# B&R Automation Studio project NAELD004C00R10L518F00 (part 12)

#### Act_OptP0930MagConv1FB.st
```iecst
ACTION Act_OptP0930MagConv1FB:

	//Magazine Conveyor
	IF tyP0930MagConv1.tyFB.tyBtnStop.bRtCompl = TRUE THEN
		eMagConv2Clp1Act	:= MagConv2ClpActStop;

		IF p_eMagConv2Clp1Stat = MagConv2ClpActStop AND p_eMagConv2Clp1Status = Done THEN
			eMagConv2Clp1Act	:= MagConv2ClpActIdle;

			tyP0930MagConv1.tyFB.tyBtnEnt.bRtCompl	:= FALSE;
			tyP0930MagConv1.tyFB.tyBtnEnt.bValue	:= FALSE;
			tyP0930MagConv1.tyFB.tyBtnEnt.bRtLk		:= FALSE;

			tyP0930MagConv1.tyFB.tyBtnExit.bRtCompl	:= FALSE;
			tyP0930MagConv1.tyFB.tyBtnExit.bValue	:= FALSE;
			tyP0930MagConv1.tyFB.tyBtnExit.bRtLk	:= FALSE;

			tyP0930MagConv1.tyFB.tyBtnStop.bRtCompl	:= FALSE;
			tyP0930MagConv1.tyFB.tyBtnStop.bValue	:= TRUE;
			tyP0930MagConv1.tyFB.tyBtnStop.bRtLk	:= TRUE;
		END_IF

	ELSIF tyP0930MagConv1.tyFB.tyBtnEnt.bRtCompl = TRUE THEN
		tyP0930MagConv1.tyFB.tyBtnEnt.bValue	:= TRUE;
		tyP0930MagConv1.tyFB.tyBtnEnt.bRtLk		:= TRUE;

		tyP0930MagConv1.tyFB.tyBtnStop.bValue	:= FALSE;
		tyP0930MagConv1.tyFB.tyBtnStop.bRtLk	:= FALSE;

		eMagConv2Clp1Act	:= MagConv2ClpActEnt;

		IF p_eMagConv2Clp1Stat = MagConv2ClpActEnt AND p_eMagConv2Clp1Status = Done THEN
			eMagConv2Clp1Act	:= MagConv2ClpActIdle;

			tyP0930MagConv1.tyFB.tyBtnEnt.bRtCompl	:= FALSE;

			tyP0930MagConv1.tyFB.tyBtnEnt.bValue	:= FALSE;
			tyP0930MagConv1.tyFB.tyBtnEnt.bRtLk		:= FALSE;

			tyP0930MagConv1.tyFB.tyBtnStop.bValue	:= TRUE;
			tyP0930MagConv1.tyFB.tyBtnStop.bRtLk	:= TRUE;
		END_IF

	ELSIF (p_eMagConv2Clp1Stat = MagConv2ClpActPreExit AND p_eMagConv2Clp1Status = Done) THEN
		eMagConv2Clp1Act	:= MagConv2ClpActIdle;

		tyP0930MagConv1.tyFB.tyBtnExit.bRtCompl	:= FALSE;

		tyP0930MagConv1.tyFB.tyBtnExit.bValue	:= FALSE;
		tyP0930MagConv1.tyFB.tyBtnExit.bRtLk	:= FALSE;

		tyP0930MagConv1.tyFB.tyBtnStop.bValue	:= TRUE;
		tyP0930MagConv1.tyFB.tyBtnStop.bRtLk	:= TRUE;

	ELSIF (p_eMagConv2Clp1Stat = MagConv2ClpActExit AND p_eMagConv2Clp1Status = Done) THEN
		eMagConv2Clp1Act	:= MagConv2ClpActIdle;

		tyP0930MagConv1.tyFB.tyBtnExit.bRtCompl	:= FALSE;

		tyP0930MagConv1.tyFB.tyBtnExit.bValue	:= FALSE;
		tyP0930MagConv1.tyFB.tyBtnExit.bRtLk	:= FALSE;

		tyP0930MagConv1.tyFB.tyBtnStop.bValue	:= TRUE;
		tyP0930MagConv1.tyFB.tyBtnStop.bRtLk	:= TRUE;

	ELSIF tyP0930MagConv1.tyFB.tyBtnExit.bRtCompl = TRUE THEN
		tyP0930MagConv1.tyFB.tyBtnExit.bRtCompl	:= FALSE;
		tyP0930MagConv1.tyFB.tyBtnExit.bValue	:= TRUE;
		tyP0930MagConv1.tyFB.tyBtnExit.bRtLk	:= TRUE;

		tyP0930MagConv1.tyFB.tyBtnStop.bValue	:= FALSE;
		tyP0930MagConv1.tyFB.tyBtnStop.bRtLk	:= FALSE;

		IF p_tyDI.bMagConvEntSen1  THEN
			eMagConv2Clp1Act	:= MagConv2ClpActExit;
		ELSE
			IF p_tyDI.bMagPresentSen1 THEN
				eMagConv2Clp1Act	:= MagConv2ClpActPreExit;
			ELSE
				eMagConv2Clp1Act	:= MagConv2ClpActExit;
			END_IF
		END_IF
	END_IF

	//Magazine Clamper
	IF tyP0930MagConv1.tyCom.tyBtnSwitch.bValue = FALSE THEN

		//Fixed/Bottom
		IF tyP0930MagConv1.tyFB.tyBtnFixedUnclamp.bRtCompl = TRUE THEN
			tyP0930MagConv1.tyFB.tyBtnFixedUnclamp.bRtCompl	:= FALSE;

			tyP0930MagConv1.tyFB.tyBtnFixedUnclamp.bValue	:= TRUE;
			tyP0930MagConv1.tyFB.tyBtnFixedClamp.bValue		:= FALSE;

		ELSIF tyP0930MagConv1.tyFB.tyBtnFixedClamp.bRtCompl = TRUE THEN
			tyP0930MagConv1.tyFB.tyBtnFixedClamp.bRtCompl	:= FALSE;

			tyP0930MagConv1.tyFB.tyBtnFixedClamp.bValue		:= TRUE;
			tyP0930MagConv1.tyFB.tyBtnFixedUnclamp.bValue	:= FALSE;

		END_IF

		//Remote/Top
		IF tyP0930MagConv1.tyFB.tyBtnRemoteUnclamp.bRtCompl = TRUE THEN
			tyP0930MagConv1.tyFB.tyBtnRemoteUnclamp.bRtCompl	:= FALSE;

			tyP0930MagConv1.tyFB.tyBtnRemoteUnclamp.bValue	:= TRUE;
			tyP0930MagConv1.tyFB.tyBtnRemoteClamp.bValue	:= FALSE;

		ELSIF tyP0930MagConv1.tyFB.tyBtnRemoteClamp.bRtCompl = TRUE THEN
			tyP0930MagConv1.tyFB.tyBtnRemoteClamp.bRtCompl	:= FALSE;

			tyP0930MagConv1.tyFB.tyBtnRemoteClamp.bValue	:= TRUE;
			tyP0930MagConv1.tyFB.tyBtnRemoteUnclamp.bValue	:= FALSE;

		END_IF

		//Selection
		IF tyP0930MagConv1.tyFB.tyBtnSelUnclamp.bRtCompl = TRUE THEN
			tyP0930MagConv1.tyFB.tyBtnSelUnclamp.bRtCompl	:= FALSE;

			tyP0930MagConv1.tyFB.tyBtnSelUnclamp.bValue	:= TRUE;
			tyP0930MagConv1.tyFB.tyBtnSelClamp.bValue	:= FALSE;

		ELSIF tyP0930MagConv1.tyFB.tyBtnSelClamp.bRtCompl = TRUE THEN
			tyP0930MagConv1.tyFB.tyBtnSelClamp.bRtCompl	:= FALSE;

			tyP0930MagConv1.tyFB.tyBtnSelClamp.bValue	:= TRUE;
			tyP0930MagConv1.tyFB.tyBtnSelUnclamp.bValue	:= FALSE;

		END_IF

		// Fixed Clamper
		IF tyP0930MagConv1.tyFB.tyBtnFixedUnclamp.bValue = TRUE THEN

			eMagConv2Clp1Act	:= MagConv2ClpActFixClprUnclamp;

			IF p_eMagConv2Clp1Stat = MagConv2ClpActFixClprUnclamp AND p_eMagConv2Clp1Status = Done THEN

				eMagConv2Clp1Act	:= MagConv2ClpActIdle;

				tyP0930MagConv1.tyFB.tyBtnFixedUnclamp.bValue	:= FALSE;

			ELSIF p_eMagConv2Clp1Status = Error THEN

				tyP0930MagConv1.tyFB.tyBtnFixedUnclamp.bValue	:= FALSE;

			END_IF

		ELSIF tyP0930MagConv1.tyFB.tyBtnFixedClamp.bValue = TRUE THEN
			eMagConv2Clp1Act	:= MagConv2ClpActFixClprClamp;

			IF p_eMagConv2Clp1Stat = MagConv2ClpActFixClprClamp AND p_eMagConv2Clp1Status = Done THEN

				eMagConv2Clp1Act	:= MagConv2ClpActIdle;

				tyP0930MagConv1.tyFB.tyBtnFixedClamp.bValue := FALSE;

			ELSIF p_eMagConv2Clp1Status = Error THEN
				tyP0930MagConv1.tyFB.tyBtnFixedClamp.bValue := FALSE;

			END_IF

		END_IF

		//Remote Clamper
		IF tyP0930MagConv1.tyFB.tyBtnRemoteUnclamp.bValue = TRUE THEN

			eMagConv2Clp1Act	:= MagConv2ClpActRmtClprUnclamp;

			IF p_eMagConv2Clp1Stat = MagConv2ClpActRmtClprUnclamp AND p_eMagConv2Clp1Status = Done THEN

				eMagConv2Clp1Act	:= MagConv2ClpActIdle;

				tyP0930MagConv1.tyFB.tyBtnRemoteUnclamp.bValue	:= FALSE;

			ELSIF p_eMagConv2Clp1Status = Error THEN

				tyP0930MagConv1.tyFB.tyBtnRemoteUnclamp.bValue	:= FALSE;

			END_IF

		ELSIF tyP0930MagConv1.tyFB.tyBtnRemoteClamp.bValue = TRUE THEN
			eMagConv2Clp1Act	:= MagConv2ClpActRmtClprClamp;

			IF p_eMagConv2Clp1Stat = MagConv2ClpActRmtClprClamp AND p_eMagConv2Clp1Status = Done THEN

				eMagConv2Clp1Act	:= MagConv2ClpActIdle;

				tyP0930MagConv1.tyFB.tyBtnRemoteClamp.bValue := FALSE;

			ELSIF p_eMagConv2Clp1Status = Error THEN
				tyP0930MagConv1.tyFB.tyBtnRemoteClamp.bValue := FALSE;

			END_IF

		END_IF

		//Selection Clamper
		IF tyP0930MagConv1.tyFB.tyBtnSelUnclamp.bValue = TRUE THEN

			eMagConvSelClp1Act	:= PneuActExt;

			IF p_eSelClamp1Stat = PneuActExt AND p_eSelClamp1Status = Done THEN

				eMagConvSelClp1Act	:= PneuActIdle;

				tyP0930MagConv1.tyFB.tyBtnSelUnclamp.bValue	:= FALSE;

			ELSIF p_eSelClamp1Status = Error THEN
				eMagConvSelClp1Act	:= PneuActIdle;
				tyP0930MagConv1.tyFB.tyBtnSelUnclamp.bValue	:= FALSE;

			END_IF

		ELSIF tyP0930MagConv1.tyFB.tyBtnSelClamp.bValue = TRUE THEN
			eMagConvSelClp1Act	:= PneuActRet;

			IF p_eSelClamp1Stat = PneuActRet AND p_eSelClamp1Status = Done THEN

				eMagConvSelClp1Act	:= PneuActIdle;

				tyP0930MagConv1.tyFB.tyBtnSelClamp.bValue	:= FALSE;

			ELSIF p_eSelClamp1Status = Error THEN
				eMagConvSelClp1Act	:= PneuActIdle;
				tyP0930MagConv1.tyFB.tyBtnSelClamp.bValue	:= FALSE;

			END_IF

		END_IF

		//Update Status
		tyP0930MagConv1.tyDC.tyBtnFixedUnclamp.bValue	:= NOT p_bMagConv2Clp1ClprFixClampCtrl;
		tyP0930MagConv1.tyDC.tyBtnFixedClamp.bValue		:= p_bMagConv2Clp1ClprFixClampCtrl;
		tyP0930MagConv1.tyDC.tyBtnRemoteUnclamp.bValue	:= NOT p_bMagConv2Clp1ClprRmtClampCtrl;
		tyP0930MagConv1.tyDC.tyBtnRemoteClamp.bValue	:= p_bMagConv2Clp1ClprRmtClampCtrl;

		tyP0930MagConv1.tyDC.tyBtnSelUnclamp.bRtCompl	:= FALSE;
		tyP0930MagConv1.tyDC.tyBtnSelClamp.bRtCompl		:= FALSE;
		tyP0930MagConv1.tyDC.tyBtnSelUnclamp.bValue	:= p_bSelClamp1RetCtrl;
		tyP0930MagConv1.tyDC.tyBtnSelClamp.bValue	:= p_bSelClamp1ExtCtrl;
	END_IF

	//Mask
	IF p_tyUsrMgmtCurrAccessRgt.bManualFBOnly THEN

		fUIInRtStatOff(ADR(tyP0930MagConv1.tyCom.tyBtnSwitch.uiMaskRtStat));

	ELSE

		IF p_eMagConv2Clp1Status = Error THEN

			fUIInRtStatOff(ADR(tyP0930MagConv1.tyFB.tyBtnEnt.uiMaskRtStat));
			fUIInRtStatOff(ADR(tyP0930MagConv1.tyFB.tyBtnExit.uiMaskRtStat));
			fUIInRtStatOff(ADR(tyP0930MagConv1.tyFB.tyBtnFixedClamp.uiMaskRtStat));
			fUIInRtStatOff(ADR(tyP0930MagConv1.tyFB.tyBtnFixedUnclamp.uiMaskRtStat));
			fUIInRtStatOff(ADR(tyP0930MagConv1.tyFB.tyBtnRemoteClamp.uiMaskRtStat));
			fUIInRtStatOff(ADR(tyP0930MagConv1.tyFB.tyBtnRemoteUnclamp.uiMaskRtStat));
			fUIInRtStatOff(ADR(tyP0930MagConv1.tyFB.tyBtnSelClamp.uiMaskRtStat));
			fUIInRtStatOff(ADR(tyP0930MagConv1.tyFB.tyBtnSelUnclamp.uiMaskRtStat));
			fUIInRtStatHide(ADR(tyP0930MagConv1.tyCom.tyBtnSwitch.uiMaskRtStat));

		ELSIF tyP0930MagConv1.tyFB.tyBtnEnt.bRtCompl = TRUE THEN

			fUIInRtStatHide(ADR(tyP0930MagConv1.tyFB.tyBtnEnt.uiMaskRtStat));
			fUIInRtStatOff(ADR(tyP0930MagConv1.tyFB.tyBtnExit.uiMaskRtStat));
			fUIInRtStatOff(ADR(tyP0930MagConv1.tyFB.tyBtnFixedClamp.uiMaskRtStat));
			fUIInRtStatOff(ADR(tyP0930MagConv1.tyFB.tyBtnFixedUnclamp.uiMaskRtStat));
			fUIInRtStatOff(ADR(tyP0930MagConv1.tyFB.tyBtnRemoteClamp.uiMaskRtStat));
			fUIInRtStatOff(ADR(tyP0930MagConv1.tyFB.tyBtnRemoteUnclamp.uiMaskRtStat));
			fUIInRtStatOff(ADR(tyP0930MagConv1.tyFB.tyBtnSelClamp.uiMaskRtStat));
			fUIInRtStatOff(ADR(tyP0930MagConv1.tyFB.tyBtnSelUnclamp.uiMaskRtStat));
			fUIInRtStatOff(ADR(tyP0930MagConv1.tyCom.tyBtnSwitch.uiMaskRtStat));

		ELSIF tyP0930MagConv1.tyFB.tyBtnExit.bRtCompl = TRUE THEN

			fUIInRtStatOff(ADR(tyP0930MagConv1.tyFB.tyBtnEnt.uiMaskRtStat));
			fUIInRtStatHide(ADR(tyP0930MagConv1.tyFB.tyBtnExit.uiMaskRtStat));
			fUIInRtStatOff(ADR(tyP0930MagConv1.tyFB.tyBtnFixedClamp.uiMaskRtStat));
			fUIInRtStatOff(ADR(tyP0930MagConv1.tyFB.tyBtnFixedUnclamp.uiMaskRtStat));
			fUIInRtStatOff(ADR(tyP0930MagConv1.tyFB.tyBtnRemoteClamp.uiMaskRtStat));
			fUIInRtStatOff(ADR(tyP0930MagConv1.tyFB.tyBtnRemoteUnclamp.uiMaskRtStat));
			fUIInRtStatOff(ADR(tyP0930MagConv1.tyFB.tyBtnSelClamp.uiMaskRtStat));
			fUIInRtStatOff(ADR(tyP0930MagConv1.tyFB.tyBtnSelUnclamp.uiMaskRtStat));
			fUIInRtStatOff(ADR(tyP0930MagConv1.tyCom.tyBtnSwitch.uiMaskRtStat));

		ELSIF tyP0930MagConv1.tyFB.tyBtnFixedClamp.bValue = TRUE OR tyP0930MagConv1.tyFB.tyBtnRemoteClamp.bValue = TRUE
			OR tyP0930MagConv1.tyFB.tyBtnFixedUnclamp.bValue = TRUE OR tyP0930MagConv1.tyFB.tyBtnRemoteUnclamp.bValue = TRUE
			OR tyP0930MagConv1.tyFB.tyBtnSelUnclamp.bValue = TRUE OR tyP0930MagConv1.tyFB.tyBtnSelClamp.bValue = TRUE
			THEN

			fUIInRtStatOff(ADR(tyP0930MagConv1.tyFB.tyBtnEnt.uiMaskRtStat));
			fUIInRtStatOff(ADR(tyP0930MagConv1.tyFB.tyBtnExit.uiMaskRtStat));
			fUIInRtStatHide(ADR(tyP0930MagConv1.tyFB.tyBtnFixedClamp.uiMaskRtStat));
			fUIInRtStatHide(ADR(tyP0930MagConv1.tyFB.tyBtnFixedUnclamp.uiMaskRtStat));
			fUIInRtStatHide(ADR(tyP0930MagConv1.tyFB.tyBtnRemoteClamp.uiMaskRtStat));
			fUIInRtStatHide(ADR(tyP0930MagConv1.tyFB.tyBtnRemoteUnclamp.uiMaskRtStat));
			fUIInRtStatHide(ADR(tyP0930MagConv1.tyFB.tyBtnSelClamp.uiMaskRtStat));
			fUIInRtStatHide(ADR(tyP0930MagConv1.tyFB.tyBtnSelUnclamp.uiMaskRtStat));
			fUIInRtStatOff(ADR(tyP0930MagConv1.tyCom.tyBtnSwitch.uiMaskRtStat));

		ELSE

			fUIInRtStatHide(ADR(tyP0930MagConv1.tyFB.tyBtnEnt.uiMaskRtStat));
			fUIInRtStatHide(ADR(tyP0930MagConv1.tyFB.tyBtnExit.uiMaskRtStat));
			fUIInRtStatHide(ADR(tyP0930MagConv1.tyFB.tyBtnFixedClamp.uiMaskRtStat));
			fUIInRtStatHide(ADR(tyP0930MagConv1.tyFB.tyBtnFixedUnclamp.uiMaskRtStat));
			fUIInRtStatHide(ADR(tyP0930MagConv1.tyFB.tyBtnRemoteClamp.uiMaskRtStat));
			fUIInRtStatHide(ADR(tyP0930MagConv1.tyFB.tyBtnRemoteUnclamp.uiMaskRtStat));
			fUIInRtStatHide(ADR(tyP0930MagConv1.tyFB.tyBtnSelClamp.uiMaskRtStat));
			fUIInRtStatHide(ADR(tyP0930MagConv1.tyFB.tyBtnSelUnclamp.uiMaskRtStat));
			fUIInRtStatHide(ADR(tyP0930MagConv1.tyCom.tyBtnSwitch.uiMaskRtStat));

		END_IF
	END_IF

	IF p_tyDI.bMagConvCAB717MagSen1 THEN
		fUIInRtStatOff(ADR(tyP0930MagConv1.tyFB.tyBtnSelClamp.uiMaskRtStat));
	END_IF

END_ACTION
```

#### Act_OptP0930MagConv1FBStat.st
```iecst
ACTION Act_OptP0930MagConv1FBStat:

IF tyP0930MagConv1.tyFB.tyBtnFixedClamp.bValue = TRUE OR tyP0930MagConv1.tyFB.tyBtnRemoteClamp.bValue = TRUE
	OR tyP0930MagConv1.tyFB.tyBtnFixedUnclamp.bValue = TRUE OR tyP0930MagConv1.tyFB.tyBtnRemoteUnclamp.bValue = TRUE
		THEN
		tyP0930MagConv1.tyFB.tyStringStat.sValue	:= p_sMagConv2Clp1StatTxt;
ELSIF tyP0930MagConv1.tyFB.tyBtnSelUnclamp.bValue = TRUE OR tyP0930MagConv1.tyFB.tyBtnSelClamp.bValue = TRUE
		THEN
		tyP0930MagConv1.tyFB.tyStringStat.sValue	:= p_sSelClamp1StatTxt;
END_IF

END_ACTION
```

#### Act_OptP0930MagConv1Sen.st
```iecst
ACTION Act_OptP0930MagConv1Sen:

	tyP0930MagConv1.tyCom.tyBtnMagPresentSen.bValue			:= p_tyDI.bMagPresentSen1;
	tyP0930MagConv1.tyCom.tyBtnMagConvEntSen.bValue			:= p_tyDI.bMagConvEntSen1;
	tyP0930MagConv1.tyCom.tyBtnMagAIVPosSen1.bValue			:= p_tyDI.bMag1AGVInPosSen1;
	tyP0930MagConv1.tyCom.tyBtnMagAIVPosSen2.bValue			:= p_tyDI.bMag1AGVInPosSen2;
	tyP0930MagConv1.tyCom.tyBtnMagOrientationChkSen1.bValue	:= p_tyDI.bMag1OrientChkSen1;
	tyP0930MagConv1.tyCom.tyBtnMagOrientationChkSen2.bValue	:= p_tyDI.bMag1OrientChkSen2;

	tyP0930MagConv1.tyCom.tyBtnFixedClampRS.bValue			:= p_tyDI.bMag1FixedClampRS;
	tyP0930MagConv1.tyCom.tyBtnFixedUnclampRS.bValue		:= p_tyDI.bMag1FixedUnclampRS;
	tyP0930MagConv1.tyCom.tyBtnRemoteClampRS.bValue			:= p_tyDI.bMag1RemoteClampRS;
	tyP0930MagConv1.tyCom.tyBtnRemoteUnclampRS.bValue		:= p_tyDI.bMag1RemoteUnclampRS;

	tyP0930MagConv1.tyCom.tyBtnSelUnclampRS.bValue			:= p_tyDI.bMag1SelUnClampRS;

	tyP0930MagConv1.tyCom.tyBtnCAB717Sen.bValue				:= p_tyDI.bMagConvCAB717MagSen1;
	tyP0930MagConv1.tyCom.tyBtnHeightSen.bValue				:= p_tyDI.bMagConvHeightSen1 OR p_tyDI.bHighMagDetSen1;
	tyP0930MagConv1.tyCom.tyBtnMagSmallSen.bValue			:= p_tyDI.bMagConvSmallMagSen1;
	tyP0930MagConv1.tyCom.tyBtnMagLargeSen.bValue			:= p_tyDI.bMagConvLargeMagSen1;

	tyP0930MagConv1.tyCom.tyBtnMagDetSen.bValue				:= p_tyDI.bMag1FixedSideDetect;
	tyP0930MagConv1.tyCom.tyBtnSltLckSen.bValue				:= p_tyDI.bSlotLckSenMag1;

	//Machine Bitmap //17
	IF p_tyNtParamCurr.eProjMag = LDMagDual AND p_tyNtParamCurr.bMagAutoVerifyPrep = FALSE THEN
		IF tyP0930MagConv1.tyFB.tyBtnFixedClamp.bRtCompl
			OR tyP0930MagConv1.tyDC.tyBtnFixedClamp.bRtCompl THEN

			tyP0930MagConv1.tyCom.tyBitmapMc.uiValueIdx	:= 44;

		ELSIF tyP0930MagConv1.tyFB.tyBtnFixedUnclamp.bRtCompl
			OR tyP0930MagConv1.tyDC.tyBtnFixedUnclamp.bRtCompl THEN

			tyP0930MagConv1.tyCom.tyBitmapMc.uiValueIdx	:= 43;

		ELSIF tyP0930MagConv1.tyFB.tyBtnRemoteClamp.bRtCompl
			OR tyP0930MagConv1.tyDC.tyBtnRemoteClamp.bRtCompl THEN

			tyP0930MagConv1.tyCom.tyBitmapMc.uiValueIdx	:= 49;

		ELSIF tyP0930MagConv1.tyFB.tyBtnRemoteUnclamp.bRtCompl
			OR tyP0930MagConv1.tyDC.tyBtnRemoteUnclamp.bRtCompl THEN

			tyP0930MagConv1.tyCom.tyBitmapMc.uiValueIdx	:= 48;

		ELSIF tyP0930MagConv1.tyFB.tyBtnEnt.bRtCompl OR tyP0930MagConv1.tyFB.tyBtnExit.bRtCompl OR tyP0930MagConv1.tyFB.tyBtnStop.bRtCompl
			OR tyP0930MagConv1.tyDC.tyBtnMagIn.bRtCompl OR tyP0930MagConv1.tyDC.tyBtnMagOut.bRtCompl OR tyP0930MagConv1.tyDC.tyBtnStop.bRtCompl THEN

			tyP0930MagConv1.tyCom.tyBitmapMc.uiValueIdx	:= 42;

		END_IF
	ELSIF p_tyNtParamCurr.eProjMag = LDMagDual AND p_tyNtParamCurr.bMagAutoVerifyPrep THEN
		IF tyP0930MagConv1.tyFB.tyBtnFixedClamp.bRtCompl
			OR tyP0930MagConv1.tyDC.tyBtnFixedClamp.bRtCompl THEN

			tyP0930MagConv1.tyCom.tyBitmapMc.uiValueIdx	:= 2;

		ELSIF tyP0930MagConv1.tyFB.tyBtnFixedUnclamp.bRtCompl
			OR tyP0930MagConv1.tyDC.tyBtnFixedUnclamp.bRtCompl THEN

			tyP0930MagConv1.tyCom.tyBitmapMc.uiValueIdx	:= 1;

		ELSIF tyP0930MagConv1.tyFB.tyBtnRemoteClamp.bRtCompl
			 OR tyP0930MagConv1.tyDC.tyBtnRemoteClamp.bRtCompl THEN

			tyP0930MagConv1.tyCom.tyBitmapMc.uiValueIdx	:= 20;

		ELSIF tyP0930MagConv1.tyFB.tyBtnRemoteUnclamp.bRtCompl
			OR tyP0930MagConv1.tyDC.tyBtnRemoteUnclamp.bRtCompl THEN

			tyP0930MagConv1.tyCom.tyBitmapMc.uiValueIdx	:= 19;

		ELSIF tyP0930MagConv1.tyFB.tyBtnSelClamp.bRtCompl
			OR tyP0930MagConv1.tyDC.tyBtnSelClamp.bRtCompl THEN

			tyP0930MagConv1.tyCom.tyBitmapMc.uiValueIdx	:= 16;

		ELSIF tyP0930MagConv1.tyFB.tyBtnSelUnclamp.bRtCompl
			OR tyP0930MagConv1.tyDC.tyBtnSelUnclamp.bRtCompl THEN

			tyP0930MagConv1.tyCom.tyBitmapMc.uiValueIdx	:= 15;

		ELSIF tyP0930MagConv1.tyFB.tyBtnEnt.bRtCompl OR tyP0930MagConv1.tyFB.tyBtnExit.bRtCompl OR tyP0930MagConv1.tyFB.tyBtnStop.bRtCompl
			OR tyP0930MagConv1.tyDC.tyBtnMagIn.bRtCompl OR tyP0930MagConv1.tyDC.tyBtnMagOut.bRtCompl OR tyP0930MagConv1.tyDC.tyBtnStop.bRtCompl THEN

			tyP0930MagConv1.tyCom.tyBitmapMc.uiValueIdx	:= 0;

		END_IF
	ELSIF p_tyNtParamCurr.eProjMag = LDMagTriple AND p_tyNtParamCurr.bProjCurtainSenPrep = FALSE AND p_tyNtParamCurr.eCustomerReq <> Siemens AND p_tyNtParamCurr.eCustomerReq <> We_Fabricate THEN
		IF tyP0930MagConv1.tyFB.tyBtnFixedClamp.bRtCompl
			OR tyP0930MagConv1.tyDC.tyBtnFixedClamp.bRtCompl THEN

			tyP0930MagConv1.tyCom.tyBitmapMc.uiValueIdx	:= 2;

		ELSIF tyP0930MagConv1.tyFB.tyBtnFixedUnclamp.bRtCompl
			OR tyP0930MagConv1.tyDC.tyBtnFixedUnclamp.bRtCompl THEN

			tyP0930MagConv1.tyCom.tyBitmapMc.uiValueIdx	:= 1;

		ELSIF tyP0930MagConv1.tyFB.tyBtnRemoteClamp.bRtCompl
			OR tyP0930MagConv1.tyDC.tyBtnRemoteClamp.bRtCompl THEN

			tyP0930MagConv1.tyCom.tyBitmapMc.uiValueIdx	:= 16;

		ELSIF tyP0930MagConv1.tyFB.tyBtnRemoteUnclamp.bRtCompl
			OR tyP0930MagConv1.tyDC.tyBtnRemoteUnclamp.bRtCompl THEN

			tyP0930MagConv1.tyCom.tyBitmapMc.uiValueIdx	:= 15;

		ELSIF tyP0930MagConv1.tyFB.tyBtnSelClamp.bRtCompl
			OR tyP0930MagConv1.tyDC.tyBtnSelClamp.bRtCompl THEN

			tyP0930MagConv1.tyCom.tyBitmapMc.uiValueIdx	:= 22;

		ELSIF tyP0930MagConv1.tyFB.tyBtnSelUnclamp.bRtCompl
			OR tyP0930MagConv1.tyDC.tyBtnSelUnclamp.bRtCompl THEN

			tyP0930MagConv1.tyCom.tyBitmapMc.uiValueIdx	:= 21;

		ELSIF tyP0930MagConv1.tyFB.tyBtnEnt.bRtCompl OR tyP0930MagConv1.tyFB.tyBtnExit.bRtCompl OR tyP0930MagConv1.tyFB.tyBtnStop.bRtCompl
			OR tyP0930MagConv1.tyDC.tyBtnMagIn.bRtCompl OR tyP0930MagConv1.tyDC.tyBtnMagOut.bRtCompl OR tyP0930MagConv1.tyDC.tyBtnStop.bRtCompl THEN

			tyP0930MagConv1.tyCom.tyBitmapMc.uiValueIdx	:= 0;

		END_IF
	ELSIF p_tyNtParamCurr.eProjMag = LDMagTriple AND p_tyNtParamCurr.bProjCurtainSenPrep OR p_tyNtParamCurr.eCustomerReq = Siemens OR p_tyNtParamCurr.eCustomerReq = We_Fabricate THEN
		tyP0930MagConv1.tyCom.tyBitmapMc.uiValueIdx	:= 384-17;

	ELSIF p_tyNtParamCurr.eProjMag = LDMagQuadruple AND p_tyNtParamCurr.bMagAutoVerifyPrep THEN
		IF tyP0930MagConv1.tyFB.tyBtnFixedClamp.bRtCompl
			OR tyP0930MagConv1.tyDC.tyBtnFixedClamp.bRtCompl THEN

			tyP0930MagConv1.tyCom.tyBitmapMc.uiValueIdx	:= 68;

		ELSIF tyP0930MagConv1.tyFB.tyBtnFixedUnclamp.bRtCompl
			OR tyP0930MagConv1.tyDC.tyBtnFixedUnclamp.bRtCompl THEN

			tyP0930MagConv1.tyCom.tyBitmapMc.uiValueIdx	:= 67;

		ELSIF tyP0930MagConv1.tyFB.tyBtnRemoteClamp.bRtCompl
			OR tyP0930MagConv1.tyDC.tyBtnRemoteClamp.bRtCompl THEN

			tyP0930MagConv1.tyCom.tyBitmapMc.uiValueIdx	:= 70;

		ELSIF tyP0930MagConv1.tyFB.tyBtnRemoteUnclamp.bRtCompl
			OR tyP0930MagConv1.tyDC.tyBtnRemoteUnclamp.bRtCompl THEN

			tyP0930MagConv1.tyCom.tyBitmapMc.uiValueIdx	:= 69;

		ELSIF tyP0930MagConv1.tyFB.tyBtnSelClamp.bRtCompl
			OR tyP0930MagConv1.tyDC.tyBtnSelClamp.bRtCompl THEN

			tyP0930MagConv1.tyCom.tyBitmapMc.uiValueIdx	:= 72;

		ELSIF tyP0930MagConv1.tyFB.tyBtnSelUnclamp.bRtCompl
			OR tyP0930MagConv1.tyDC.tyBtnSelUnclamp.bRtCompl THEN

			tyP0930MagConv1.tyCom.tyBitmapMc.uiValueIdx	:= 71;

		ELSIF tyP0930MagConv1.tyFB.tyBtnEnt.bRtCompl OR tyP0930MagConv1.tyFB.tyBtnExit.bRtCompl OR tyP0930MagConv1.tyFB.tyBtnStop.bRtCompl
			OR tyP0930MagConv1.tyDC.tyBtnMagIn.bRtCompl OR tyP0930MagConv1.tyDC.tyBtnMagOut.bRtCompl OR tyP0930MagConv1.tyDC.tyBtnStop.bRtCompl THEN

			tyP0930MagConv1.tyCom.tyBitmapMc.uiValueIdx	:= 66;

		END_IF
	END_IF

	IF p_tyNtParamCurr.eProjMag = LDMagDual AND p_tyNtParamCurr.bMagAutoVerifyPrep = FALSE THEN
		IF tyP0930MagConv1.tyCom.tyBitmapMc.uiValueIdx < 100 THEN
			IF p_tyNtParamCurr.sJobNo = '2023-0276A01' THEN // no longer belt type //17 base
				tyP0930MagConv1.tyCom.tyBitmapMc.uiValueIdx	:= 493-17;
			ELSIF p_tyNtParamCurr.sJobNo = '2023-0258A01' THEN
				tyP0930MagConv1.tyCom.tyBitmapMc.uiValueIdx	:= 463-17;
			ELSE
				tyP0930MagConv1.tyCom.tyBitmapMc.uiValueIdx	:= tyP0930MagConv1.tyCom.tyBitmapMc.uiValueIdx + 100;
			END_IF
		END_IF
	ELSIF p_tyNtParamCurr.eProjMag = LDMagTriple AND p_tyNtParamCurr.bMagAutoVerifyPrep = FALSE AND p_tyNtParamCurr.bProjMotorizedPullerPrep = FALSE THEN
		IF tyP0930MagConv1.tyCom.tyBitmapMc.uiValueIdx < 100 THEN
			tyP0930MagConv1.tyCom.tyBitmapMc.uiValueIdx	:= tyP0930MagConv1.tyCom.tyBitmapMc.uiValueIdx + 100;
		END_IF
	ELSIF p_tyNtParamCurr.eProjMag = LDMagDual AND p_tyNtParamCurr.bMagAutoVerifyPrep = TRUE THEN
		IF tyP0930MagConv1.tyCom.tyBitmapMc.uiValueIdx < 200 THEN
			tyP0930MagConv1.tyCom.tyBitmapMc.uiValueIdx	:= tyP0930MagConv1.tyCom.tyBitmapMc.uiValueIdx + 200;
		END_IF
	ELSIF p_tyNtParamCurr.eProjMag = LDMagTriple AND p_tyNtParamCurr.bMagAutoVerifyPrep = FALSE AND p_tyNtParamCurr.bProjMotorizedPullerPrep = TRUE THEN
		IF tyP0930MagConv1.tyCom.tyBitmapMc.uiValueIdx < 300 THEN
			tyP0930MagConv1.tyCom.tyBitmapMc.uiValueIdx	:= tyP0930MagConv1.tyCom.tyBitmapMc.uiValueIdx + 300;
		END_IF
	END_IF

END_ACTION
```

#### Act_OptP0930Navi.st
```iecst
ACTION Act_OptP0930Navi:

	CASE p_tyNtParamCurr.eProjMag OF
		LDMagDual:
			IF tyP0930MagConv1.tyNavi2Lyr1.tyBtnBack.bRtCompl = TRUE THEN
				tyP0930MagConv1.tyNavi2Lyr1.tyBtnBack.bRtCompl	:= FALSE;
				tyP0930MagConv1.tyNavi2Lyr1.tyBtnBack.bValue	:= FALSE;

				eChgPage	:= UIP0920MtrNPneuCtrl;
				bDispMagConv1	:= TRUE;
				bDispMagConv2	:= FALSE;
				bDispMagConv3	:= FALSE;
				bDispMagConv4	:= FALSE;

			ELSIF tyP0930MagConv1.tyNavi2Lyr1.tyBtnLeft.bRtCompl = TRUE OR tyP0930MagConv1.tyNavi2Lyr1.tyBtnRgt.bRtCompl = TRUE THEN
				tyP0930MagConv1.tyNavi2Lyr1.tyBtnLeft.bRtCompl			:= FALSE;
				tyP0930MagConv1.tyNavi2Lyr1.tyBtnLeft.bValue			:= FALSE;
				tyP0930MagConv1.tyNavi2Lyr1.tyBtnRgt.bRtCompl			:= FALSE;
				tyP0930MagConv1.tyNavi2Lyr1.tyBtnRgt.bValue				:= FALSE;
				eChgPage												:= UIP0931MagConv2;
				bDispMagConv1	:= FALSE;
				bDispMagConv2	:= TRUE;
				bDispMagConv3	:= FALSE;
				bDispMagConv4	:= FALSE;
			END_IF

		LDMagTriple:
			IF tyP0930MagConv1.tyNavi3Lyr1.tyBtnBack.bRtCompl = TRUE THEN
				tyP0930MagConv1.tyNavi3Lyr1.tyBtnBack.bRtCompl	:= FALSE;
				tyP0930MagConv1.tyNavi3Lyr1.tyBtnBack.bValue	:= FALSE;

				eChgPage	:= UIP0920MtrNPneuCtrl;
				bDispMagConv1	:= TRUE;
				bDispMagConv2	:= FALSE;
				bDispMagConv3	:= FALSE;
				bDispMagConv4	:= FALSE;

			ELSIF tyP0930MagConv1.tyNavi3Lyr1.tyBtnLeft.bRtCompl = TRUE THEN
				tyP0930MagConv1.tyNavi3Lyr1.tyBtnLeft.bRtCompl			:= FALSE;
				tyP0930MagConv1.tyNavi3Lyr1.tyBtnLeft.bValue			:= FALSE;
				eChgPage												:= UIP0932MagConv3;
				bDispMagConv1	:= FALSE;
				bDispMagConv2	:= FALSE;
				bDispMagConv3	:= TRUE;
				bDispMagConv4	:= FALSE;

			ELSIF tyP0930MagConv1.tyNavi3Lyr1.tyBtnRgt.bRtCompl = TRUE THEN
				tyP0930MagConv1.tyNavi3Lyr1.tyBtnRgt.bRtCompl			:= FALSE;
				tyP0930MagConv1.tyNavi3Lyr1.tyBtnRgt.bValue				:= FALSE;
				eChgPage												:= UIP0931MagConv2;
				bDispMagConv1	:= FALSE;
				bDispMagConv2	:= TRUE;
				bDispMagConv3	:= FALSE;
				bDispMagConv4	:= FALSE;
			END_IF

		LDMagQuadruple:
			IF tyP0930MagConv1.tyNavi4Lyr1.tyBtnBack.bRtCompl = TRUE THEN
				tyP0930MagConv1.tyNavi4Lyr1.tyBtnBack.bRtCompl	:= FALSE;
				tyP0930MagConv1.tyNavi4Lyr1.tyBtnBack.bValue	:= FALSE;

				eChgPage	:= UIP0920MtrNPneuCtrl;
				bDispMagConv1	:= TRUE;
				bDispMagConv2	:= FALSE;
				bDispMagConv3	:= FALSE;
				bDispMagConv4	:= FALSE;

			ELSIF tyP0930MagConv1.tyNavi4Lyr1.tyBtnLeft.bRtCompl = TRUE THEN
				tyP0930MagConv1.tyNavi4Lyr1.tyBtnLeft.bRtCompl			:= FALSE;
				tyP0930MagConv1.tyNavi4Lyr1.tyBtnLeft.bValue			:= FALSE;
				eChgPage												:= UIP0939MagConv4;
				bDispMagConv1	:= FALSE;
				bDispMagConv2	:= FALSE;
				bDispMagConv3	:= FALSE;
				bDispMagConv4	:= TRUE;

			ELSIF tyP0930MagConv1.tyNavi4Lyr1.tyBtnRgt.bRtCompl = TRUE THEN
				tyP0930MagConv1.tyNavi4Lyr1.tyBtnRgt.bRtCompl			:= FALSE;
				tyP0930MagConv1.tyNavi4Lyr1.tyBtnRgt.bValue				:= FALSE;
				eChgPage												:= UIP0931MagConv2;
				bDispMagConv1	:= FALSE;
				bDispMagConv2	:= TRUE;
				bDispMagConv3	:= FALSE;
				bDispMagConv4	:= FALSE;

			END_IF
	END_CASE

END_ACTION
```

#### Act_OptP0930RstMnl.st
```iecst
ACTION Act_OptP0930RstMnl:

	IF EDGEPOS((bManualMod = FALSE) OR (p_eMagConv2Clp1Status = Error)) THEN

		eMagConv2Clp1Act	:= MagConv2ClpActIdle;
		eMagConvSelClp1Act	:= PneuActIdle;
		//Magazine Conveyor
		//FB
		tyP0930MagConv1.tyFB.tyBtnEnt.bRtCompl				:= FALSE;
		tyP0930MagConv1.tyFB.tyBtnExit.bRtCompl				:= FALSE;
		tyP0930MagConv1.tyFB.tyBtnStop.bRtCompl				:= FALSE;

		tyP0930MagConv1.tyFB.tyBtnEnt.bValue				:= FALSE;
		tyP0930MagConv1.tyFB.tyBtnExit.bValue				:= FALSE;
		tyP0930MagConv1.tyFB.tyBtnStop.bValue				:= TRUE;

		tyP0930MagConv1.tyFB.tyBtnEnt.bRtLk					:= FALSE;
		tyP0930MagConv1.tyFB.tyBtnExit.bRtLk				:= FALSE;
		tyP0930MagConv1.tyFB.tyBtnStop.bRtLk				:= TRUE;

		tyP0930MagConv1.tyFB.tyBtnEnt.uiMaskRtStat.0		:= TRUE;
		tyP0930MagConv1.tyFB.tyBtnExit.uiMaskRtStat.0		:= TRUE;
		tyP0930MagConv1.tyCom.tyBtnSwitch.uiMaskRtStat.0	:= TRUE;

		//Direct
		tyP0930MagConv1.tyDC.tyBtnMagIn.bRtCompl			:= FALSE;
		tyP0930MagConv1.tyDC.tyBtnMagOut.bRtCompl			:= FALSE;
		tyP0930MagConv1.tyDC.tyBtnStop.bRtCompl				:= FALSE;

		tyP0930MagConv1.tyDC.tyBtnMagIn.bValue				:= FALSE;
		tyP0930MagConv1.tyDC.tyBtnMagOut.bValue				:= FALSE;
		tyP0930MagConv1.tyDC.tyBtnStop.bValue				:= TRUE;

		tyP0930MagConv1.tyDC.tyBtnMagIn.bRtLk				:= FALSE;
		tyP0930MagConv1.tyDC.tyBtnMagOut.bRtLk				:= FALSE;
		tyP0930MagConv1.tyDC.tyBtnStop.bRtLk				:= TRUE;

		tyP0930MagConv1.tyDC.tyBtnMagIn.uiMaskRtStat.0		:= TRUE;
		tyP0930MagConv1.tyDC.tyBtnMagOut.uiMaskRtStat.0		:= TRUE;
		tyP0930MagConv1.tyCom.tyBtnSwitch.uiMaskRtStat.0	:= TRUE;

		//Magazine Clamper
		//FB
		//Fixed/Bottom
		tyP0930MagConv1.tyFB.tyBtnFixedClamp.bRtCompl			:= FALSE;
		tyP0930MagConv1.tyFB.tyBtnFixedUnclamp.bRtCompl			:= FALSE;

		tyP0930MagConv1.tyFB.tyBtnFixedClamp.bValue				:= FALSE;
		tyP0930MagConv1.tyFB.tyBtnFixedUnclamp.bValue			:= FALSE;

		//Remote/Top
		tyP0930MagConv1.tyFB.tyBtnRemoteClamp.bRtCompl			:= FALSE;
		tyP0930MagConv1.tyFB.tyBtnRemoteUnclamp.bRtCompl		:= FALSE;

		tyP0930MagConv1.tyFB.tyBtnRemoteClamp.bValue			:= FALSE;
		tyP0930MagConv1.tyFB.tyBtnRemoteUnclamp.bValue			:= FALSE;

		//Selection
		tyP0930MagConv1.tyFB.tyBtnSelClamp.bRtCompl			:= FALSE;
		tyP0930MagConv1.tyFB.tyBtnSelUnclamp.bRtCompl		:= FALSE;

		tyP0930MagConv1.tyFB.tyBtnSelClamp.bValue			:= FALSE;
		tyP0930MagConv1.tyFB.tyBtnSelUnclamp.bValue			:= FALSE;

		tyP0930MagConv1.tyFB.tyBtnFixedClamp.uiMaskRtStat.0		:= TRUE;
		tyP0930MagConv1.tyFB.tyBtnFixedUnclamp.uiMaskRtStat.0	:= TRUE;
		tyP0930MagConv1.tyFB.tyBtnRemoteClamp.uiMaskRtStat.0	:= TRUE;
		tyP0930MagConv1.tyFB.tyBtnRemoteUnclamp.uiMaskRtStat.0	:= TRUE;
		tyP0930MagConv1.tyFB.tyBtnSelClamp.uiMaskRtStat.0		:= TRUE;
		tyP0930MagConv1.tyFB.tyBtnSelUnclamp.uiMaskRtStat.0		:= TRUE;

		tyP0930MagConv1.tyCom.tyBtnSwitch.uiMaskRtStat.0		:= TRUE;

		//Direct
		//Fixed/Bottom
		tyP0930MagConv1.tyDC.tyBtnFixedClamp.bRtCompl			:= FALSE;
		tyP0930MagConv1.tyDC.tyBtnFixedUnclamp.bRtCompl			:= FALSE;

		tyP0930MagConv1.tyDC.tyBtnFixedClamp.bValue				:= FALSE;
		tyP0930MagConv1.tyDC.tyBtnFixedUnclamp.bValue			:= FALSE;

		//Remote/Top
		tyP0930MagConv1.tyDC.tyBtnRemoteClamp.bRtCompl			:= FALSE;
		tyP0930MagConv1.tyDC.tyBtnRemoteUnclamp.bRtCompl		:= FALSE;

		tyP0930MagConv1.tyDC.tyBtnRemoteClamp.bValue			:= FALSE;
		tyP0930MagConv1.tyDC.tyBtnRemoteUnclamp.bValue			:= FALSE;

		//Selection
		tyP0930MagConv1.tyDC.tyBtnSelClamp.bRtCompl				:= FALSE;
		tyP0930MagConv1.tyDC.tyBtnSelUnclamp.bRtCompl			:= FALSE;

		tyP0930MagConv1.tyDC.tyBtnSelClamp.bValue				:= FALSE;
		tyP0930MagConv1.tyDC.tyBtnSelUnclamp.bValue				:= FALSE;

		tyP0930MagConv1.tyDC.tyBtnFixedClamp.uiMaskRtStat.0		:= TRUE;
		tyP0930MagConv1.tyDC.tyBtnFixedUnclamp.uiMaskRtStat.0	:= TRUE;
		tyP0930MagConv1.tyDC.tyBtnRemoteClamp.uiMaskRtStat.0	:= TRUE;
		tyP0930MagConv1.tyDC.tyBtnRemoteUnclamp.uiMaskRtStat.0	:= TRUE;
		tyP0930MagConv1.tyDC.tyBtnSelClamp.uiMaskRtStat.0		:= TRUE;
		tyP0930MagConv1.tyDC.tyBtnSelUnclamp.uiMaskRtStat.0		:= TRUE;

		tyP0930MagConv1.tyCom.tyBtnSwitch.uiMaskRtStat.0		:= TRUE;

	END_IF

	IF EDGEPOS(bManualMod = FALSE) THEN
		tyP0930MagConv1.tyCom.tyBtnSwitch.bValue := FALSE;

		IF p_tyNtParamCurr.bMagAutoVerifyPrep = FALSE THEN
			fUIInRtStatHide(ADR(tyP0930MagConv1.tyDC.tyLyrWithoutSelClamp.uiRtStat));
			fUIInRtStatOff(ADR(tyP0930MagConv1.tyFB.tyLyrWithoutSelClamp.uiRtStat));
		ELSE

			fUIInRtStatHide(ADR(tyP0930MagConv1.tyDC.tyLyr.uiRtStat));
			fUIInRtStatOff(ADR(tyP0930MagConv1.tyFB.tyLyr.uiRtStat));
		END_IF
	END_IF

END_ACTION
```

#### Act_EntP0931Disp.st
```iecst
ACTION Act_EntP0931Disp:

	//Access Address
	p_tyC0002FullMask ACCESS ADR(tyP0931MagConv2.tyFullMaskHide);

//	p_tyC0004Navi ACCESS ADR(tyP0931MagConv2.tyNaviBack);
	CASE p_tyNtParamCurr.eProjMag OF
		LDMagDual:
			p_tyC0004Navi ACCESS ADR(tyP0931MagConv2.tyNavi2Lyr2);
		LDMagTriple:
			p_tyC0004Navi ACCESS ADR(tyP0931MagConv2.tyNavi3Lyr2);
		LDMagQuadruple:
			p_tyC0004Navi ACCESS ADR(tyP0931MagConv2.tyNavi4Lyr2);
	END_CASE

	p_tyC0005Main ACCESS ADR(tyCommon.tyMain);

	p_tyC0007Notif ACCESS ADR(tyCommon.tyNotif);

	p_tyC0008MsgBox ACCESS ADR(tyP0931MagConv2.tyMsgBoxHide);

	p_tyC0009Info ACCESS ADR(tyCommon.tyInfo);

	p_tyP0931Mag2ConvCom ACCESS ADR(tyP0931MagConv2.tyCom);
	p_tyP0931Mag2ConvDC ACCESS ADR(tyP0931MagConv2.tyDC);
	p_tyP0931Mag2ConvFB ACCESS ADR(tyP0931MagConv2.tyFB);

	IF p_tyNtParamCurr.eProjMag = LDMagDual AND p_tyNtParamCurr.bMagAutoVerifyPrep = FALSE THEN
		tyP0931MagConv2.tyCom.tyBitmapMc.usiValueIdx	:= 142;
	ELSIF p_tyNtParamCurr.eProjMag = LDMagDual AND p_tyNtParamCurr.bMagAutoVerifyPrep = TRUE THEN
		tyP0931MagConv2.tyCom.tyBitmapMc.usiValueIdx	:= 200;
	ELSIF p_tyNtParamCurr.eProjMag = LDMagTriple AND p_tyNtParamCurr.bMagAutoVerifyPrep = TRUE THEN
		tyP0931MagConv2.tyCom.tyBitmapMc.usiValueIdx	:= 0;
	ELSIF p_tyNtParamCurr.eProjMag = LDMagQuadruple AND p_tyNtParamCurr.bMagAutoVerifyPrep = TRUE THEN
		tyP0931MagConv2.tyCom.tyBitmapMc.usiValueIdx	:= 70;
	ELSE
		tyP0931MagConv2.tyCom.tyBitmapMc.usiValueIdx	:= 100;
	END_IF

	IF p_tyNtParamCurr.bMagAutoVerifyPrep = FALSE THEN
		tyP0931MagConv2.tyFB.tyBtnFixedClamp.usiTxtIdx	:= 6;
		tyP0931MagConv2.tyFB.tyBtnFixedUnclamp.usiTxtIdx:= 6;
		tyP0931MagConv2.tyFB.tyBtnRemoteClamp.usiTxtIdx	:= 6;
		tyP0931MagConv2.tyFB.tyBtnRemoteUnclamp.usiTxtIdx:= 6;
	ELSE
		tyP0931MagConv2.tyFB.tyBtnFixedClamp.usiTxtIdx	:= 6;
		tyP0931MagConv2.tyFB.tyBtnFixedUnclamp.usiTxtIdx:= 6;
		tyP0931MagConv2.tyFB.tyBtnRemoteClamp.usiTxtIdx	:= 6;
		tyP0931MagConv2.tyFB.tyBtnRemoteUnclamp.usiTxtIdx:= 6;

	END_IF

	IF p_tyNtParamCurr.bMagAutoVerifyPrep = FALSE THEN
		IF tyP0931MagConv2.tyCom.tyBtnSwitch.bValue THEN
			fUIInRtStatHide(ADR(tyP0931MagConv2.tyFB.tyLyr.uiRtStat));
			fUIInRtStatHide(ADR(tyP0931MagConv2.tyDC.tyLyr.uiRtStat));
			fUIInRtStatHide(ADR(tyP0931MagConv2.tyFB.tyLyrWithoutSelClamp.uiRtStat));
			fUIInRtStatOff(ADR(tyP0931MagConv2.tyDC.tyLyrWithoutSelClamp.uiRtStat));
		ELSE
			fUIInRtStatHide(ADR(tyP0931MagConv2.tyFB.tyLyr.uiRtStat));
			fUIInRtStatHide(ADR(tyP0931MagConv2.tyDC.tyLyr.uiRtStat));
			fUIInRtStatOff(ADR(tyP0931MagConv2.tyFB.tyLyrWithoutSelClamp.uiRtStat));
			fUIInRtStatHide(ADR(tyP0931MagConv2.tyDC.tyLyrWithoutSelClamp.uiRtStat));
		END_IF
	ELSE
		IF tyP0931MagConv2.tyCom.tyBtnSwitch.bValue THEN
			fUIInRtStatHide(ADR(tyP0931MagConv2.tyFB.tyLyr.uiRtStat));
			fUIInRtStatOff(ADR(tyP0931MagConv2.tyDC.tyLyr.uiRtStat));
			fUIInRtStatHide(ADR(tyP0931MagConv2.tyFB.tyLyrWithoutSelClamp.uiRtStat));
			fUIInRtStatHide(ADR(tyP0931MagConv2.tyDC.tyLyrWithoutSelClamp.uiRtStat));
		ELSE
			fUIInRtStatOff(ADR(tyP0931MagConv2.tyFB.tyLyr.uiRtStat));
			fUIInRtStatHide(ADR(tyP0931MagConv2.tyDC.tyLyr.uiRtStat));
			fUIInRtStatHide(ADR(tyP0931MagConv2.tyFB.tyLyrWithoutSelClamp.uiRtStat));
			fUIInRtStatHide(ADR(tyP0931MagConv2.tyDC.tyLyrWithoutSelClamp.uiRtStat));
		END_IF
	END_IF

END_ACTION
```

#### Act_OptP0931FullMask.st
```iecst
ACTION Act_OptP0931FullMask:

	IF eCurrPage = UIP0931MagConv2 THEN

		IF p_tyDI.bEStopSig = FALSE THEN
			p_tyC0002FullMask ACCESS ADR(tyP0931MagConv2.tyFullMaskEStop);

		ELSIF p_tyDI.bCoverSWSig = FALSE THEN
			p_tyC0002FullMask ACCESS ADR(tyP0931MagConv2.tyFullMaskCWSig);

		ELSIF p_tyDI.bSafetyRlySig = FALSE THEN
			p_tyC0002FullMask ACCESS ADR(tyP0931MagConv2.tyFullMaskSafetyRly);

		ELSE
			p_tyC0002FullMask ACCESS ADR(tyP0931MagConv2.tyFullMaskHide);

		END_IF

	END_IF

END_ACTION
```

#### Act_OptP0931MagConv2ChgLyr.st
```iecst
ACTION Act_OptP0931MagConv2ChgLyr:

	IF p_tyNtParamCurr.bMagAutoVerifyPrep THEN
		IF tyP0931MagConv2.tyCom.tyBtnSwitch.bRtCompl THEN
			tyP0931MagConv2.tyCom.tyBtnSwitch.bRtCompl	:= FALSE;

			IF tyP0931MagConv2.tyCom.tyBtnSwitch.bValue = TRUE THEN
				fUIInRtStatOff(ADR(tyP0931MagConv2.tyDC.tyLyr.uiRtStat));
				fUIInRtStatHide(ADR(tyP0931MagConv2.tyFB.tyLyr.uiRtStat));
			ELSE
				fUIInRtStatHide(ADR(tyP0931MagConv2.tyDC.tyLyr.uiRtStat));
				fUIInRtStatOff(ADR(tyP0931MagConv2.tyFB.tyLyr.uiRtStat));
			END_IF

		END_IF
	ELSE
		IF tyP0931MagConv2.tyCom.tyBtnSwitch.bRtCompl THEN
			tyP0931MagConv2.tyCom.tyBtnSwitch.bRtCompl	:= FALSE;

			IF tyP0931MagConv2.tyCom.tyBtnSwitch.bValue = TRUE THEN
				fUIInRtStatOff(ADR(tyP0931MagConv2.tyDC.tyLyrWithoutSelClamp.uiRtStat));
				fUIInRtStatHide(ADR(tyP0931MagConv2.tyFB.tyLyrWithoutSelClamp.uiRtStat));
			ELSE
				fUIInRtStatHide(ADR(tyP0931MagConv2.tyDC.tyLyrWithoutSelClamp.uiRtStat));
				fUIInRtStatOff(ADR(tyP0931MagConv2.tyFB.tyLyrWithoutSelClamp.uiRtStat));
			END_IF

		END_IF
	END_IF

END_ACTION
```

#### Act_OptP0931MagConv2DC.st
```iecst
ACTION Act_OptP0931MagConv2DC:

	//Magazine Conveyor
	IF tyP0931MagConv2.tyDC.tyBtnStop.bRtCompl = TRUE THEN
		eMagConv2Clp2Act	:= MagConv2ClpActStop;

		IF p_eMagConv2Clp2Stat = MagConv2ClpActStop AND p_eMagConv2Clp2Status = Done THEN
			eMagConv2Clp2Act	:= MagConv2ClpActIdle;

			tyP0931MagConv2.tyDC.tyBtnStop.bRtCompl		:= FALSE;
			tyP0931MagConv2.tyDC.tyBtnStop.bValue		:= TRUE;
			tyP0931MagConv2.tyDC.tyBtnStop.bRtLk		:= TRUE;

			tyP0931MagConv2.tyDC.tyBtnMagIn.bRtCompl	:= FALSE;
			tyP0931MagConv2.tyDC.tyBtnMagIn.bValue		:= FALSE;
			tyP0931MagConv2.tyDC.tyBtnMagIn.bRtLk		:= FALSE;

			tyP0931MagConv2.tyDC.tyBtnMagOut.bRtCompl	:= FALSE;
			tyP0931MagConv2.tyDC.tyBtnMagOut.bValue		:= FALSE;
			tyP0931MagConv2.tyDC.tyBtnMagOut.bRtLk		:= FALSE;
		END_IF

	ELSIF tyP0931MagConv2.tyDC.tyBtnMagIn.bRtCompl = TRUE THEN
		tyP0931MagConv2.tyDC.tyBtnMagIn.bValue	:= TRUE;
		tyP0931MagConv2.tyDC.tyBtnMagIn.bRtLk	:= TRUE;

		tyP0931MagConv2.tyDC.tyBtnStop.bValue	:= FALSE;
		tyP0931MagConv2.tyDC.tyBtnStop.bRtLk	:= FALSE;

		IF p_tyNtParamCurr.eProjMagConvDir = ConvDirLToR OR p_tyNtParamCurr.eProjMagConvDir = ConvDirLToL THEN

			eMagConv2Clp2Act	:= MagConv2ClpActSetMtrSigOnOrLToR;

			IF p_eMagConv2Clp2Stat = MagConv2ClpActSetMtrSigOnOrLToR AND p_eMagConv2Clp2Status = Done THEN
				eMagConv2Clp2Act	:= MagConv2ClpActIdle;

				tyP0931MagConv2.tyDC.tyBtnMagIn.bRtCompl	:= FALSE;
			END_IF

		ELSE

			eMagConv2Clp2Act	:= MagConv2ClpActSetMtrDirOrRToL;

			IF p_eMagConv2Clp2Stat = MagConv2ClpActSetMtrDirOrRToL AND p_eMagConv2Clp2Status = Done THEN
				eMagConv2Clp2Act	:= MagConv2ClpActIdle;

				tyP0931MagConv2.tyDC.tyBtnMagIn.bRtCompl	:= FALSE;
			END_IF

		END_IF

	ELSIF tyP0931MagConv2.tyDC.tyBtnMagOut.bRtCompl = TRUE THEN
		tyP0931MagConv2.tyDC.tyBtnMagOut.bValue	:= TRUE;
		tyP0931MagConv2.tyDC.tyBtnMagOut.bRtLk	:= TRUE;

		tyP0931MagConv2.tyDC.tyBtnStop.bValue	:= FALSE;
		tyP0931MagConv2.tyDC.tyBtnStop.bRtLk	:= FALSE;

		IF p_tyNtParamCurr.eProjMagConvDir = ConvDirLToR OR p_tyNtParamCurr.eProjMagConvDir = ConvDirRToR THEN

			eMagConv2Clp2Act	:= MagConv2ClpActSetMtrSigOnOrLToR;

			IF p_eMagConv2Clp2Stat = MagConv2ClpActSetMtrSigOnOrLToR AND p_eMagConv2Clp2Status = Done THEN
				eMagConv2Clp2Act	:= MagConv2ClpActIdle;

				tyP0931MagConv2.tyDC.tyBtnMagOut.bRtCompl	:= FALSE;
			END_IF

		ELSE

			eMagConv2Clp2Act	:= MagConv2ClpActSetMtrDirOrRToL;

			IF p_eMagConv2Clp2Stat = MagConv2ClpActSetMtrDirOrRToL AND p_eMagConv2Clp2Status = Done THEN
				eMagConv2Clp2Act	:= MagConv2ClpActIdle;

				tyP0931MagConv2.tyDC.tyBtnMagOut.bRtCompl	:= FALSE;
			END_IF

		END_IF

	END_IF

	//Magazine Clamper
	IF tyP0931MagConv2.tyCom.tyBtnSwitch.bValue = TRUE THEN
		IF p_bSelClamp2TwoCtrlOut = FALSE THEN
			IF tyP0931MagConv2.tyDC.tyBtnSelUnclamp.bRtCompl = TRUE THEN
				tyP0931MagConv2.tyDC.tyBtnSelUnclamp.bValue := TRUE;
				tyP0931MagConv2.tyDC.tyBtnSelClamp.bValue := FALSE;

				eMagConvSelClp2Act	:= PneuActSetExt;

				IF p_eSelClamp2Stat = PneuActSetExt AND p_eSelClamp2Status = Done THEN
					eMagConvSelClp2Act	:= PneuActIdle;

					tyP0931MagConv2.tyDC.tyBtnSelUnclamp.bRtCompl	:= FALSE;
				END_IF

			ELSIF tyP0931MagConv2.tyDC.tyBtnSelClamp.bRtCompl = TRUE THEN
				tyP0931MagConv2.tyDC.tyBtnSelClamp.bValue := TRUE;
				tyP0931MagConv2.tyDC.tyBtnSelUnclamp.bValue := FALSE;

				eMagConvSelClp2Act	:= PneuActSetRet;

				IF p_eSelClamp2Stat = PneuActSetRet AND p_eSelClamp2Status = Done THEN
					eMagConvSelClp2Act	:= PneuActIdle;

					tyP0931MagConv2.tyDC.tyBtnSelClamp.bRtCompl	:= FALSE;
				END_IF
			END_IF

		ELSE
			IF (tyP0931MagConv2.tyDC.tyBtnSelUnclamp.bRtCompl = TRUE) OR (tyP0931MagConv2.tyDC.tyBtnSelClamp.bRtCompl = TRUE) THEN
				IF (tyP0931MagConv2.tyDC.tyBtnSelUnclamp.bValue = TRUE) AND (tyP0931MagConv2.tyDC.tyBtnSelClamp.bValue = TRUE) THEN
					eMagConvSelClp2Act	:= PneuActSetAll;

					IF p_eSelClamp2Stat = PneuActSetAll AND p_eSelClamp2Status = Done THEN
						eMagConvSelClp2Act	:= PneuActIdle;

						tyP0931MagConv2.tyDC.tyBtnSelUnclamp.bRtCompl		:= FALSE;
						tyP0931MagConv2.tyDC.tyBtnSelClamp.bRtCompl			:= FALSE;
					END_IF

				ELSIF (tyP0931MagConv2.tyDC.tyBtnSelUnclamp.bValue = TRUE) AND (tyP0931MagConv2.tyDC.tyBtnSelClamp.bValue = FALSE) THEN
					eMagConvSelClp2Act	:= PneuActSetExt;

					IF p_eSelClamp2Stat = PneuActSetExt AND p_eSelClamp2Status = Done THEN
						eMagConvSelClp2Act	:= PneuActIdle;

						tyP0931MagConv2.tyDC.tyBtnSelUnclamp.bRtCompl		:= FALSE;
						tyP0931MagConv2.tyDC.tyBtnSelClamp.bRtCompl			:= FALSE;
					END_IF

				ELSIF (tyP0931MagConv2.tyDC.tyBtnSelUnclamp.bValue = FALSE) AND (tyP0931MagConv2.tyDC.tyBtnSelClamp.bValue = TRUE) THEN
					eMagConvSelClp2Act	:= PneuActSetRet;

					IF p_eSelClamp2Stat = PneuActSetRet AND p_eSelClamp2Status = Done THEN
						eMagConvSelClp2Act	:= PneuActIdle;

						tyP0931MagConv2.tyDC.tyBtnSelUnclamp.bRtCompl		:= FALSE;
						tyP0931MagConv2.tyDC.tyBtnSelClamp.bRtCompl			:= FALSE;
					END_IF

				ELSE
					eMagConvSelClp2Act	:= PneuActRstAll;

					IF p_eSelClamp2Stat = PneuActRstAll AND p_eSelClamp2Status = Done THEN
						eMagConvSelClp2Act	:= PneuActIdle;

						tyP0931MagConv2.tyDC.tyBtnSelUnclamp.bRtCompl		:= FALSE;
						tyP0931MagConv2.tyDC.tyBtnSelClamp.bRtCompl			:= FALSE;
					END_IF

				END_IF
			END_IF
		END_IF

		IF p_bMagConv2Clp1ClprTwoOutputCtrl = FALSE THEN

			//Fixed
			IF tyP0931MagConv2.tyDC.tyBtnFixedClamp.bRtCompl = TRUE THEN
				tyP0931MagConv2.tyDC.tyBtnFixedClamp.bValue		:= TRUE;
				tyP0931MagConv2.tyDC.tyBtnFixedUnclamp.bValue	:= FALSE;

				eMagConv2Clp2Act	:= MagConv2ClpActFixClprSetClamp;

				IF p_eMagConv2Clp2Stat = MagConv2ClpActFixClprSetClamp AND p_eMagConv2Clp2Status = Done THEN
					eMagConv2Clp2Act	:= MagConv2ClpActIdle;

					tyP0931MagConv2.tyDC.tyBtnFixedClamp.bRtCompl	:= FALSE;
				END_IF

			ELSIF tyP0931MagConv2.tyDC.tyBtnFixedUnclamp.bRtCompl = TRUE THEN
				tyP0931MagConv2.tyDC.tyBtnFixedUnclamp.bValue	:= TRUE;
				tyP0931MagConv2.tyDC.tyBtnFixedClamp.bValue		:= FALSE;

				eMagConv2Clp2Act	:= MagConv2ClpActFixClprSetUnclamp;

				IF p_eMagConv2Clp2Stat = MagConv2ClpActFixClprSetUnclamp AND p_eMagConv2Clp2Status = Done THEN
					eMagConv2Clp2Act	:= MagConv2ClpActIdle;

					tyP0931MagConv2.tyDC.tyBtnFixedUnclamp.bRtCompl	:= FALSE;
				END_IF

			END_IF

			//Remote
			IF tyP0931MagConv2.tyDC.tyBtnRemoteClamp.bRtCompl = TRUE THEN
				tyP0931MagConv2.tyDC.tyBtnRemoteClamp.bValue		:= TRUE;
				tyP0931MagConv2.tyDC.tyBtnRemoteUnclamp.bValue		:= FALSE;

				eMagConv2Clp2Act	:= MagConv2ClpActRmtClprSetClamp;

				IF p_eMagConv2Clp2Stat = MagConv2ClpActRmtClprSetClamp AND p_eMagConv2Clp2Status = Done THEN
					eMagConv2Clp2Act	:= MagConv2ClpActIdle;

					tyP0931MagConv2.tyDC.tyBtnRemoteClamp.bRtCompl	:= FALSE;
				END_IF

			ELSIF tyP0931MagConv2.tyDC.tyBtnRemoteUnclamp.bRtCompl = TRUE THEN
				tyP0931MagConv2.tyDC.tyBtnRemoteUnclamp.bValue	:= TRUE;
				tyP0931MagConv2.tyDC.tyBtnRemoteClamp.bValue	:= FALSE;

				eMagConv2Clp2Act	:= MagConv2ClpActRmtClprSetUnclamp;

				IF p_eMagConv2Clp2Stat = MagConv2ClpActRmtClprSetUnclamp AND p_eMagConv2Clp2Status = Done THEN
					eMagConv2Clp2Act	:= MagConv2ClpActIdle;

					tyP0931MagConv2.tyDC.tyBtnRemoteUnclamp.bRtCompl	:= FALSE;
				END_IF

			END_IF

		ELSE

			//Fixed
			IF (tyP0931MagConv2.tyDC.tyBtnFixedClamp.bRtCompl = TRUE) OR (tyP0931MagConv2.tyDC.tyBtnFixedUnclamp.bRtCompl = TRUE) THEN

				IF (tyP0931MagConv2.tyDC.tyBtnFixedClamp.bValue = TRUE) AND (tyP0931MagConv2.tyDC.tyBtnFixedUnclamp.bValue = TRUE) THEN

					eMagConv2Clp2Act	:= MagConv2ClpActFixClprSetAll;

					IF p_eMagConv2Clp2Stat = MagConv2ClpActFixClprSetAll AND p_eMagConv2Clp2Status = Done THEN

						eMagConv2Clp2Act	:= MagConv2ClpActIdle;

						tyP0931MagConv2.tyDC.tyBtnFixedClamp.bRtCompl	:= FALSE;
						tyP0931MagConv2.tyDC.tyBtnFixedUnclamp.bRtCompl	:= FALSE;
					END_IF

				ELSIF (tyP0931MagConv2.tyDC.tyBtnFixedClamp.bValue = TRUE) AND (tyP0931MagConv2.tyDC.tyBtnFixedUnclamp.bValue = FALSE) THEN
					eMagConv2Clp2Act	:= MagConv2ClpActFixClprSetClamp;

					IF p_eMagConv2Clp2Stat = MagConv2ClpActFixClprSetClamp AND p_eMagConv2Clp2Status = Done THEN

						eMagConv2Clp2Act	:= MagConv2ClpActIdle;

						tyP0931MagConv2.tyDC.tyBtnFixedClamp.bRtCompl	:= FALSE;
						tyP0931MagConv2.tyDC.tyBtnFixedUnclamp.bRtCompl	:= FALSE;
					END_IF

				ELSIF (tyP0931MagConv2.tyDC.tyBtnFixedClamp.bValue = FALSE) AND (tyP0931MagConv2.tyDC.tyBtnFixedUnclamp.bValue = TRUE) THEN
					eMagConv2Clp2Act	:= MagConv2ClpActFixClprSetUnclamp;

					IF p_eMagConv2Clp2Stat = MagConv2ClpActFixClprSetUnclamp AND p_eMagConv2Clp2Status = Done THEN

						eMagConv2Clp2Act	:= MagConv2ClpActIdle;

						tyP0931MagConv2.tyDC.tyBtnFixedClamp.bRtCompl	:= FALSE;
						tyP0931MagConv2.tyDC.tyBtnFixedUnclamp.bRtCompl	:= FALSE;
					END_IF

				ELSE
					eMagConv2Clp2Act	:= MagConv2ClpActFixClprRstAll;

					IF p_eMagConv2Clp2Stat = MagConv2ClpActFixClprRstAll AND p_eMagConv2Clp2Status = Done THEN

						eMagConv2Clp2Act	:= MagConv2ClpActIdle;

						tyP0931MagConv2.tyDC.tyBtnFixedClamp.bRtCompl	:= FALSE;
						tyP0931MagConv2.tyDC.tyBtnFixedUnclamp.bRtCompl	:= FALSE;
					END_IF

				END_IF

				//Remote
				IF (tyP0931MagConv2.tyDC.tyBtnRemoteClamp.bRtCompl = TRUE) OR (tyP0931MagConv2.tyDC.tyBtnRemoteUnclamp.bRtCompl = TRUE) THEN

					IF (tyP0931MagConv2.tyDC.tyBtnRemoteClamp.bValue = TRUE) AND (tyP0931MagConv2.tyDC.tyBtnRemoteUnclamp.bValue = TRUE) THEN

						eMagConv2Clp2Act	:= MagConv2ClpActRmtClprSetAll;

						IF p_eMagConv2Clp2Stat = MagConv2ClpActRmtClprSetAll AND p_eMagConv2Clp2Status = Done THEN

							eMagConv2Clp2Act	:= MagConv2ClpActIdle;

							tyP0931MagConv2.tyDC.tyBtnRemoteClamp.bRtCompl		:= FALSE;
							tyP0931MagConv2.tyDC.tyBtnRemoteUnclamp.bRtCompl	:= FALSE;
						END_IF

					ELSIF (tyP0931MagConv2.tyDC.tyBtnRemoteClamp.bValue = TRUE) AND (tyP0931MagConv2.tyDC.tyBtnRemoteUnclamp.bValue = FALSE) THEN
						eMagConv2Clp2Act	:= MagConv2ClpActRmtClprSetClamp;

						IF p_eMagConv2Clp2Stat = MagConv2ClpActRmtClprSetClamp AND p_eMagConv2Clp2Status = Done THEN

							eMagConv2Clp2Act	:= MagConv2ClpActIdle;

							tyP0931MagConv2.tyDC.tyBtnRemoteClamp.bRtCompl	:= FALSE;
							tyP0931MagConv2.tyDC.tyBtnRemoteUnclamp.bRtCompl	:= FALSE;
						END_IF

					ELSIF (tyP0931MagConv2.tyDC.tyBtnRemoteClamp.bValue = FALSE) AND (tyP0931MagConv2.tyDC.tyBtnRemoteUnclamp.bValue = TRUE) THEN
						eMagConv2Clp2Act	:= MagConv2ClpActRmtClprSetUnclamp;

						IF p_eMagConv2Clp2Stat = MagConv2ClpActRmtClprSetUnclamp AND p_eMagConv2Clp2Status = Done THEN

							eMagConv2Clp2Act	:= MagConv2ClpActIdle;

							tyP0931MagConv2.tyDC.tyBtnRemoteClamp.bRtCompl	:= FALSE;
							tyP0931MagConv2.tyDC.tyBtnRemoteUnclamp.bRtCompl	:= FALSE;
						END_IF

					ELSE
						eMagConv2Clp2Act	:= MagConv2ClpActRmtClprRstAll;

						IF p_eMagConv2Clp2Stat = MagConv2ClpActRmtClprRstAll AND p_eMagConv2Clp2Status = Done THEN

							eMagConv2Clp2Act	:= MagConv2ClpActIdle;

							tyP0931MagConv2.tyDC.tyBtnRemoteClamp.bRtCompl	:= FALSE;
							tyP0931MagConv2.tyDC.tyBtnRemoteUnclamp.bRtCompl	:= FALSE;
						END_IF

					END_IF
				END_IF

			END_IF

		END_IF

		//Fixed
		tyP0931MagConv2.tyFB.tyBtnFixedClamp.bRtCompl		:= FALSE;
		tyP0931MagConv2.tyFB.tyBtnFixedClamp.bValue			:= FALSE;
		tyP0931MagConv2.tyFB.tyBtnFixedUnclamp.bRtCompl		:= FALSE;
		tyP0931MagConv2.tyFB.tyBtnFixedUnclamp.bValue		:= FALSE;
		tyP0931MagConv2.tyFB.tyBtnSelClamp.bRtCompl			:= FALSE;
		tyP0931MagConv2.tyFB.tyBtnSelClamp.bValue			:= FALSE;

		//Remote
		tyP0931MagConv2.tyFB.tyBtnRemoteClamp.bRtCompl		:= FALSE;
		tyP0931MagConv2.tyFB.tyBtnRemoteClamp.bValue		:= FALSE;
		tyP0931MagConv2.tyFB.tyBtnRemoteUnclamp.bRtCompl	:= FALSE;
		tyP0931MagConv2.tyFB.tyBtnRemoteUnclamp.bValue		:= FALSE;

	END_IF

	//Mask
	IF p_eMagConv2Clp2Status = Error THEN

		fUIInRtStatOff(ADR(tyP0931MagConv2.tyDC.tyBtnMagIn.uiMaskRtStat));
		fUIInRtStatOff(ADR(tyP0931MagConv2.tyDC.tyBtnMagOut.uiMaskRtStat));
		fUIInRtStatOff(ADR(tyP0931MagConv2.tyDC.tyBtnFixedClamp.uiMaskRtStat));
		fUIInRtStatOff(ADR(tyP0931MagConv2.tyDC.tyBtnFixedUnclamp.uiMaskRtStat));
		fUIInRtStatOff(ADR(tyP0931MagConv2.tyDC.tyBtnRemoteClamp.uiMaskRtStat));
		fUIInRtStatOff(ADR(tyP0931MagConv2.tyDC.tyBtnRemoteUnclamp.uiMaskRtStat));

	ELSIF tyP0931MagConv2.tyDC.tyBtnMagIn.bValue = TRUE THEN

		fUIInRtStatHide(ADR(tyP0931MagConv2.tyDC.tyBtnMagIn.uiMaskRtStat));
		fUIInRtStatOff(ADR(tyP0931MagConv2.tyDC.tyBtnMagOut.uiMaskRtStat));
		fUIInRtStatOff(ADR(tyP0931MagConv2.tyDC.tyBtnFixedClamp.uiMaskRtStat));
		fUIInRtStatOff(ADR(tyP0931MagConv2.tyDC.tyBtnFixedUnclamp.uiMaskRtStat));
		fUIInRtStatOff(ADR(tyP0931MagConv2.tyDC.tyBtnRemoteClamp.uiMaskRtStat));
		fUIInRtStatOff(ADR(tyP0931MagConv2.tyDC.tyBtnRemoteUnclamp.uiMaskRtStat));

	ELSIF tyP0931MagConv2.tyDC.tyBtnMagOut.bValue = TRUE THEN

		fUIInRtStatOff(ADR(tyP0931MagConv2.tyDC.tyBtnMagIn.uiMaskRtStat));
		fUIInRtStatHide(ADR(tyP0931MagConv2.tyDC.tyBtnMagOut.uiMaskRtStat));
		fUIInRtStatOff(ADR(tyP0931MagConv2.tyDC.tyBtnFixedClamp.uiMaskRtStat));
		fUIInRtStatOff(ADR(tyP0931MagConv2.tyDC.tyBtnFixedUnclamp.uiMaskRtStat));
		fUIInRtStatOff(ADR(tyP0931MagConv2.tyDC.tyBtnRemoteClamp.uiMaskRtStat));
		fUIInRtStatOff(ADR(tyP0931MagConv2.tyDC.tyBtnRemoteUnclamp.uiMaskRtStat));

	ELSE

		fUIInRtStatHide(ADR(tyP0931MagConv2.tyDC.tyBtnMagIn.uiMaskRtStat));
		fUIInRtStatHide(ADR(tyP0931MagConv2.tyDC.tyBtnMagOut.uiMaskRtStat));
		fUIInRtStatHide(ADR(tyP0931MagConv2.tyDC.tyBtnFixedClamp.uiMaskRtStat));
		fUIInRtStatHide(ADR(tyP0931MagConv2.tyDC.tyBtnFixedUnclamp.uiMaskRtStat));
		fUIInRtStatHide(ADR(tyP0931MagConv2.tyDC.tyBtnRemoteClamp.uiMaskRtStat));
		fUIInRtStatHide(ADR(tyP0931MagConv2.tyDC.tyBtnRemoteUnclamp.uiMaskRtStat));

	END_IF

END_ACTION
```

#### Act_OptP0931MagConv2FB.st
```iecst
ACTION Act_OptP0931MagConv2FB:

	//Magazine Conveyor
	IF tyP0931MagConv2.tyFB.tyBtnStop.bRtCompl = TRUE THEN
		eMagConv2Clp2Act	:= MagConv2ClpActStop;

		IF p_eMagConv2Clp2Stat = MagConv2ClpActStop AND p_eMagConv2Clp2Status = Done THEN
			eMagConv2Clp2Act	:= MagConv2ClpActIdle;

			tyP0931MagConv2.tyFB.tyBtnEnt.bRtCompl	:= FALSE;
			tyP0931MagConv2.tyFB.tyBtnEnt.bValue	:= FALSE;
			tyP0931MagConv2.tyFB.tyBtnEnt.bRtLk		:= FALSE;

			tyP0931MagConv2.tyFB.tyBtnExit.bRtCompl	:= FALSE;
			tyP0931MagConv2.tyFB.tyBtnExit.bValue	:= FALSE;
			tyP0931MagConv2.tyFB.tyBtnExit.bRtLk	:= FALSE;

			tyP0931MagConv2.tyFB.tyBtnStop.bRtCompl	:= FALSE;
			tyP0931MagConv2.tyFB.tyBtnStop.bValue	:= TRUE;
			tyP0931MagConv2.tyFB.tyBtnStop.bRtLk	:= TRUE;
		END_IF

	ELSIF tyP0931MagConv2.tyFB.tyBtnEnt.bRtCompl = TRUE THEN
		tyP0931MagConv2.tyFB.tyBtnEnt.bValue	:= TRUE;
		tyP0931MagConv2.tyFB.tyBtnEnt.bRtLk		:= TRUE;

		tyP0931MagConv2.tyFB.tyBtnStop.bValue	:= FALSE;
		tyP0931MagConv2.tyFB.tyBtnStop.bRtLk	:= FALSE;

		eMagConv2Clp2Act	:= MagConv2ClpActEnt;

		IF p_eMagConv2Clp2Stat = MagConv2ClpActEnt AND p_eMagConv2Clp2Status = Done THEN
			eMagConv2Clp2Act	:= MagConv2ClpActIdle;

			tyP0931MagConv2.tyFB.tyBtnEnt.bRtCompl	:= FALSE;

			tyP0931MagConv2.tyFB.tyBtnEnt.bValue	:= FALSE;
			tyP0931MagConv2.tyFB.tyBtnEnt.bRtLk		:= FALSE;

			tyP0931MagConv2.tyFB.tyBtnStop.bValue	:= TRUE;
			tyP0931MagConv2.tyFB.tyBtnStop.bRtLk	:= TRUE;
		END_IF

	ELSIF (p_eMagConv2Clp2Stat = MagConv2ClpActPreExit AND p_eMagConv2Clp2Status = Done) THEN
		eMagConv2Clp2Act	:= MagConv2ClpActIdle;

		tyP0931MagConv2.tyFB.tyBtnExit.bRtCompl	:= FALSE;

		tyP0931MagConv2.tyFB.tyBtnExit.bValue	:= FALSE;
		tyP0931MagConv2.tyFB.tyBtnExit.bRtLk	:= FALSE;

		tyP0931MagConv2.tyFB.tyBtnStop.bValue	:= TRUE;
		tyP0931MagConv2.tyFB.tyBtnStop.bRtLk	:= TRUE;

	ELSIF (p_eMagConv2Clp2Stat = MagConv2ClpActExit AND p_eMagConv2Clp2Status = Done) THEN
		eMagConv2Clp2Act	:= MagConv2ClpActIdle;

		tyP0931MagConv2.tyFB.tyBtnExit.bRtCompl	:= FALSE;

		tyP0931MagConv2.tyFB.tyBtnExit.bValue	:= FALSE;
		tyP0931MagConv2.tyFB.tyBtnExit.bRtLk	:= FALSE;

		tyP0931MagConv2.tyFB.tyBtnStop.bValue	:= TRUE;
		tyP0931MagConv2.tyFB.tyBtnStop.bRtLk	:= TRUE;

	ELSIF tyP0931MagConv2.tyFB.tyBtnExit.bRtCompl = TRUE THEN
		tyP0931MagConv2.tyFB.tyBtnExit.bRtCompl	:= FALSE;
		tyP0931MagConv2.tyFB.tyBtnExit.bValue	:= TRUE;
		tyP0931MagConv2.tyFB.tyBtnExit.bRtLk	:= TRUE;

		tyP0931MagConv2.tyFB.tyBtnStop.bValue	:= FALSE;
		tyP0931MagConv2.tyFB.tyBtnStop.bRtLk	:= FALSE;

		IF p_tyDI.bMagConvEntSen2  THEN
			eMagConv2Clp2Act	:= MagConv2ClpActExit;
		ELSE
			IF p_tyDI.bMagPresentSen2 THEN
				eMagConv2Clp2Act	:= MagConv2ClpActPreExit;
			ELSE
				eMagConv2Clp2Act	:= MagConv2ClpActExit;
			END_IF
		END_IF
	END_IF

	//Magazine Clamper
	IF tyP0931MagConv2.tyCom.tyBtnSwitch.bValue = FALSE THEN

		//Fixed/Bottom
		IF tyP0931MagConv2.tyFB.tyBtnFixedUnclamp.bRtCompl = TRUE THEN
			tyP0931MagConv2.tyFB.tyBtnFixedUnclamp.bRtCompl	:= FALSE;

			tyP0931MagConv2.tyFB.tyBtnFixedUnclamp.bValue	:= TRUE;
			tyP0931MagConv2.tyFB.tyBtnFixedClamp.bValue		:= FALSE;

		ELSIF tyP0931MagConv2.tyFB.tyBtnFixedClamp.bRtCompl = TRUE THEN
			tyP0931MagConv2.tyFB.tyBtnFixedClamp.bRtCompl	:= FALSE;

			tyP0931MagConv2.tyFB.tyBtnFixedClamp.bValue		:= TRUE;
			tyP0931MagConv2.tyFB.tyBtnFixedUnclamp.bValue	:= FALSE;

		END_IF

		//Remote/Top
		IF tyP0931MagConv2.tyFB.tyBtnRemoteUnclamp.bRtCompl = TRUE THEN
			tyP0931MagConv2.tyFB.tyBtnRemoteUnclamp.bRtCompl	:= FALSE;

			tyP0931MagConv2.tyFB.tyBtnRemoteUnclamp.bValue	:= TRUE;
			tyP0931MagConv2.tyFB.tyBtnRemoteClamp.bValue	:= FALSE;

		ELSIF tyP0931MagConv2.tyFB.tyBtnRemoteClamp.bRtCompl = TRUE THEN
			tyP0931MagConv2.tyFB.tyBtnRemoteClamp.bRtCompl	:= FALSE;

			tyP0931MagConv2.tyFB.tyBtnRemoteClamp.bValue	:= TRUE;
			tyP0931MagConv2.tyFB.tyBtnRemoteUnclamp.bValue	:= FALSE;

		END_IF

		//Selection
		IF tyP0931MagConv2.tyFB.tyBtnSelUnclamp.bRtCompl = TRUE THEN
			tyP0931MagConv2.tyFB.tyBtnSelUnclamp.bRtCompl	:= FALSE;

			tyP0931MagConv2.tyFB.tyBtnSelUnclamp.bValue	:= TRUE;
			tyP0931MagConv2.tyFB.tyBtnSelClamp.bValue	:= FALSE;

		ELSIF tyP0931MagConv2.tyFB.tyBtnSelClamp.bRtCompl = TRUE THEN
			tyP0931MagConv2.tyFB.tyBtnSelClamp.bRtCompl	:= FALSE;

			tyP0931MagConv2.tyFB.tyBtnSelClamp.bValue	:= TRUE;
			tyP0931MagConv2.tyFB.tyBtnSelUnclamp.bValue	:= FALSE;

		END_IF

		// Fixed Clamper
		IF tyP0931MagConv2.tyFB.tyBtnFixedUnclamp.bValue = TRUE THEN

			eMagConv2Clp2Act	:= MagConv2ClpActFixClprUnclamp;

			IF p_eMagConv2Clp2Stat = MagConv2ClpActFixClprUnclamp AND p_eMagConv2Clp2Status = Done THEN

				eMagConv2Clp2Act	:= MagConv2ClpActIdle;

				tyP0931MagConv2.tyFB.tyBtnFixedUnclamp.bValue	:= FALSE;

			ELSIF p_eMagConv2Clp2Status = Error THEN

				tyP0931MagConv2.tyFB.tyBtnFixedUnclamp.bValue	:= FALSE;

			END_IF

		ELSIF tyP0931MagConv2.tyFB.tyBtnFixedClamp.bValue = TRUE THEN
			eMagConv2Clp2Act	:= MagConv2ClpActFixClprClamp;

			IF p_eMagConv2Clp2Stat = MagConv2ClpActFixClprClamp AND p_eMagConv2Clp2Status = Done THEN

				eMagConv2Clp2Act	:= MagConv2ClpActIdle;

				tyP0931MagConv2.tyFB.tyBtnFixedClamp.bValue := FALSE;

			ELSIF p_eMagConv2Clp2Status = Error THEN
				tyP0931MagConv2.tyFB.tyBtnFixedClamp.bValue := FALSE;

			END_IF

		END_IF

		//Remote Clamper
		IF tyP0931MagConv2.tyFB.tyBtnRemoteUnclamp.bValue = TRUE THEN

			eMagConv2Clp2Act	:= MagConv2ClpActRmtClprUnclamp;

			IF p_eMagConv2Clp2Stat = MagConv2ClpActRmtClprUnclamp AND p_eMagConv2Clp2Status = Done THEN

				eMagConv2Clp2Act	:= MagConv2ClpActIdle;

				tyP0931MagConv2.tyFB.tyBtnRemoteUnclamp.bValue	:= FALSE;

			ELSIF p_eMagConv2Clp2Status = Error THEN

				tyP0931MagConv2.tyFB.tyBtnRemoteUnclamp.bValue	:= FALSE;

			END_IF

		ELSIF tyP0931MagConv2.tyFB.tyBtnRemoteClamp.bValue = TRUE THEN
			eMagConv2Clp2Act	:= MagConv2ClpActRmtClprClamp;

			IF p_eMagConv2Clp2Stat = MagConv2ClpActRmtClprClamp AND p_eMagConv2Clp2Status = Done THEN

				eMagConv2Clp2Act	:= MagConv2ClpActIdle;

				tyP0931MagConv2.tyFB.tyBtnRemoteClamp.bValue := FALSE;

			ELSIF p_eMagConv2Clp2Status = Error THEN
				tyP0931MagConv2.tyFB.tyBtnRemoteClamp.bValue := FALSE;

			END_IF

		END_IF

		//Selection Clamper
		IF tyP0931MagConv2.tyFB.tyBtnSelUnclamp.bValue = TRUE THEN

			eMagConvSelClp2Act	:= PneuActExt;

			IF p_eSelClamp2Stat = PneuActExt AND p_eSelClamp2Status = Done THEN

				eMagConvSelClp2Act	:= PneuActIdle;

				tyP0931MagConv2.tyFB.tyBtnSelUnclamp.bValue	:= FALSE;

			ELSIF p_eSelClamp2Status = Error THEN
				eMagConvSelClp2Act	:= PneuActIdle;
				tyP0931MagConv2.tyFB.tyBtnSelUnclamp.bValue	:= FALSE;

			END_IF

		ELSIF tyP0931MagConv2.tyFB.tyBtnSelClamp.bValue = TRUE THEN
			eMagConvSelClp2Act	:= PneuActRet;

			IF p_eSelClamp2Stat = PneuActRet AND p_eSelClamp2Status = Done THEN

				eMagConvSelClp2Act	:= PneuActIdle;

				tyP0931MagConv2.tyFB.tyBtnSelClamp.bValue	:= FALSE;

			ELSIF p_eSelClamp2Status = Error THEN
				eMagConvSelClp2Act	:= PneuActIdle;
				tyP0931MagConv2.tyFB.tyBtnSelClamp.bValue	:= FALSE;

			END_IF

		END_IF

		//Update Status
		tyP0931MagConv2.tyDC.tyBtnFixedUnclamp.bValue	:= NOT p_bMagConv2Clp2ClprFixClampCtrl;
		tyP0931MagConv2.tyDC.tyBtnFixedClamp.bValue		:= p_bMagConv2Clp2ClprFixClampCtrl;
		tyP0931MagConv2.tyDC.tyBtnRemoteUnclamp.bValue	:= NOT p_bMagConv2Clp2ClprRmtClampCtrl;
		tyP0931MagConv2.tyDC.tyBtnRemoteClamp.bValue	:= p_bMagConv2Clp2ClprRmtClampCtrl;

		tyP0931MagConv2.tyDC.tyBtnSelUnclamp.bRtCompl	:= FALSE;
		tyP0931MagConv2.tyDC.tyBtnSelClamp.bRtCompl		:= FALSE;
		tyP0931MagConv2.tyDC.tyBtnSelUnclamp.bValue	:= p_bSelClamp2RetCtrl;
		tyP0931MagConv2.tyDC.tyBtnSelClamp.bValue	:= p_bSelClamp2ExtCtrl;
	END_IF

	//Mask
	IF p_tyUsrMgmtCurrAccessRgt.bManualFBOnly THEN

		fUIInRtStatOff(ADR(tyP0931MagConv2.tyCom.tyBtnSwitch.uiMaskRtStat));

	ELSE

		IF p_eMagConv2Clp2Status = Error THEN

			fUIInRtStatOff(ADR(tyP0931MagConv2.tyFB.tyBtnEnt.uiMaskRtStat));
			fUIInRtStatOff(ADR(tyP0931MagConv2.tyFB.tyBtnExit.uiMaskRtStat));
			fUIInRtStatOff(ADR(tyP0931MagConv2.tyFB.tyBtnFixedClamp.uiMaskRtStat));
			fUIInRtStatOff(ADR(tyP0931MagConv2.tyFB.tyBtnFixedUnclamp.uiMaskRtStat));
			fUIInRtStatOff(ADR(tyP0931MagConv2.tyFB.tyBtnRemoteClamp.uiMaskRtStat));
			fUIInRtStatOff(ADR(tyP0931MagConv2.tyFB.tyBtnRemoteUnclamp.uiMaskRtStat));
			fUIInRtStatOff(ADR(tyP0931MagConv2.tyFB.tyBtnSelClamp.uiMaskRtStat));
			fUIInRtStatOff(ADR(tyP0931MagConv2.tyFB.tyBtnSelUnclamp.uiMaskRtStat));
			fUIInRtStatHide(ADR(tyP0931MagConv2.tyCom.tyBtnSwitch.uiMaskRtStat));

		ELSIF tyP0931MagConv2.tyFB.tyBtnEnt.bRtCompl = TRUE THEN

			fUIInRtStatHide(ADR(tyP0931MagConv2.tyFB.tyBtnEnt.uiMaskRtStat));
			fUIInRtStatOff(ADR(tyP0931MagConv2.tyFB.tyBtnExit.uiMaskRtStat));
			fUIInRtStatOff(ADR(tyP0931MagConv2.tyFB.tyBtnFixedClamp.uiMaskRtStat));
			fUIInRtStatOff(ADR(tyP0931MagConv2.tyFB.tyBtnFixedUnclamp.uiMaskRtStat));
			fUIInRtStatOff(ADR(tyP0931MagConv2.tyFB.tyBtnRemoteClamp.uiMaskRtStat));
			fUIInRtStatOff(ADR(tyP0931MagConv2.tyFB.tyBtnRemoteUnclamp.uiMaskRtStat));
			fUIInRtStatOff(ADR(tyP0931MagConv2.tyFB.tyBtnSelClamp.uiMaskRtStat));
			fUIInRtStatOff(ADR(tyP0931MagConv2.tyFB.tyBtnSelUnclamp.uiMaskRtStat));
			fUIInRtStatOff(ADR(tyP0931MagConv2.tyCom.tyBtnSwitch.uiMaskRtStat));

		ELSIF tyP0931MagConv2.tyFB.tyBtnExit.bRtCompl = TRUE THEN

			fUIInRtStatOff(ADR(tyP0931MagConv2.tyFB.tyBtnEnt.uiMaskRtStat));
			fUIInRtStatHide(ADR(tyP0931MagConv2.tyFB.tyBtnExit.uiMaskRtStat));
			fUIInRtStatOff(ADR(tyP0931MagConv2.tyFB.tyBtnFixedClamp.uiMaskRtStat));
			fUIInRtStatOff(ADR(tyP0931MagConv2.tyFB.tyBtnFixedUnclamp.uiMaskRtStat));
			fUIInRtStatOff(ADR(tyP0931MagConv2.tyFB.tyBtnRemoteClamp.uiMaskRtStat));
			fUIInRtStatOff(ADR(tyP0931MagConv2.tyFB.tyBtnRemoteUnclamp.uiMaskRtStat));
			fUIInRtStatOff(ADR(tyP0931MagConv2.tyFB.tyBtnSelClamp.uiMaskRtStat));
			fUIInRtStatOff(ADR(tyP0931MagConv2.tyFB.tyBtnSelUnclamp.uiMaskRtStat));
			fUIInRtStatOff(ADR(tyP0931MagConv2.tyCom.tyBtnSwitch.uiMaskRtStat));

		ELSIF tyP0931MagConv2.tyFB.tyBtnFixedClamp.bValue = TRUE OR tyP0931MagConv2.tyFB.tyBtnRemoteClamp.bValue = TRUE
			OR tyP0931MagConv2.tyFB.tyBtnFixedUnclamp.bValue = TRUE OR tyP0931MagConv2.tyFB.tyBtnRemoteUnclamp.bValue = TRUE
			OR tyP0931MagConv2.tyFB.tyBtnSelClamp.bValue = TRUE OR tyP0931MagConv2.tyFB.tyBtnSelUnclamp.bValue = TRUE
			THEN

			fUIInRtStatOff(ADR(tyP0931MagConv2.tyFB.tyBtnEnt.uiMaskRtStat));
			fUIInRtStatOff(ADR(tyP0931MagConv2.tyFB.tyBtnExit.uiMaskRtStat));
			fUIInRtStatHide(ADR(tyP0931MagConv2.tyFB.tyBtnFixedClamp.uiMaskRtStat));
			fUIInRtStatHide(ADR(tyP0931MagConv2.tyFB.tyBtnFixedUnclamp.uiMaskRtStat));
			fUIInRtStatHide(ADR(tyP0931MagConv2.tyFB.tyBtnRemoteClamp.uiMaskRtStat));
			fUIInRtStatHide(ADR(tyP0931MagConv2.tyFB.tyBtnRemoteUnclamp.uiMaskRtStat));
			fUIInRtStatHide(ADR(tyP0931MagConv2.tyFB.tyBtnSelClamp.uiMaskRtStat));
			fUIInRtStatHide(ADR(tyP0931MagConv2.tyFB.tyBtnSelUnclamp.uiMaskRtStat));
			fUIInRtStatOff(ADR(tyP0931MagConv2.tyCom.tyBtnSwitch.uiMaskRtStat));

		ELSE

			fUIInRtStatHide(ADR(tyP0931MagConv2.tyFB.tyBtnEnt.uiMaskRtStat));
			fUIInRtStatHide(ADR(tyP0931MagConv2.tyFB.tyBtnExit.uiMaskRtStat));
			fUIInRtStatHide(ADR(tyP0931MagConv2.tyFB.tyBtnFixedClamp.uiMaskRtStat));
			fUIInRtStatHide(ADR(tyP0931MagConv2.tyFB.tyBtnFixedUnclamp.uiMaskRtStat));
			fUIInRtStatHide(ADR(tyP0931MagConv2.tyFB.tyBtnRemoteClamp.uiMaskRtStat));
			fUIInRtStatHide(ADR(tyP0931MagConv2.tyFB.tyBtnRemoteUnclamp.uiMaskRtStat));
			fUIInRtStatHide(ADR(tyP0931MagConv2.tyFB.tyBtnSelClamp.uiMaskRtStat));
			fUIInRtStatHide(ADR(tyP0931MagConv2.tyFB.tyBtnSelUnclamp.uiMaskRtStat));
			fUIInRtStatHide(ADR(tyP0931MagConv2.tyCom.tyBtnSwitch.uiMaskRtStat));

		END_IF
	END_IF

	IF p_tyDI.bMagConvCAB717MagSen2 THEN
		fUIInRtStatOff(ADR(tyP0931MagConv2.tyFB.tyBtnSelClamp.uiMaskRtStat));
	END_IF
END_ACTION
```

#### Act_OptP0931MagConv2FBStat.st
```iecst
ACTION Act_OptP0931MagConv2FBStat:

	IF tyP0931MagConv2.tyFB.tyBtnFixedClamp.bValue = TRUE OR tyP0931MagConv2.tyFB.tyBtnRemoteClamp.bValue = TRUE
		OR tyP0931MagConv2.tyFB.tyBtnFixedUnclamp.bValue = TRUE OR tyP0931MagConv2.tyFB.tyBtnRemoteUnclamp.bValue = TRUE
		THEN
		tyP0931MagConv2.tyFB.tyStringStat.sValue	:= p_sMagConv2Clp2StatTxt;
	ELSIF tyP0931MagConv2.tyFB.tyBtnSelUnclamp.bValue = TRUE OR tyP0931MagConv2.tyFB.tyBtnSelClamp.bValue = TRUE
		THEN
		tyP0931MagConv2.tyFB.tyStringStat.sValue	:= p_sSelClamp2StatTxt;
	END_IF
END_ACTION
```

#### Act_OptP0931MagConv2Sen.st
```iecst
ACTION Act_OptP0931MagConv2Sen:

	tyP0931MagConv2.tyCom.tyBtnMagPresentSen.bValue			:= p_tyDI.bMagPresentSen2;
	tyP0931MagConv2.tyCom.tyBtnMagConvEntSen.bValue			:= p_tyDI.bMagConvEntSen2;
	tyP0931MagConv2.tyCom.tyBtnMagAIVPosSen1.bValue			:= p_tyDI.bMag2AGVInPosSen1;
	tyP0931MagConv2.tyCom.tyBtnMagAIVPosSen2.bValue			:= p_tyDI.bMag2AGVInPosSen2;
	tyP0931MagConv2.tyCom.tyBtnMagOrientationChkSen1.bValue	:= p_tyDI.bMag2OrientChkSen1;
	tyP0931MagConv2.tyCom.tyBtnMagOrientationChkSen2.bValue	:= p_tyDI.bMag2OrientChkSen2;

	tyP0931MagConv2.tyCom.tyBtnFixedClampRS.bValue			:= p_tyDI.bMag2FixedClampRS;
	tyP0931MagConv2.tyCom.tyBtnFixedUnclampRS.bValue		:= p_tyDI.bMag2FixedUnclampRS;
	tyP0931MagConv2.tyCom.tyBtnRemoteClampRS.bValue			:= p_tyDI.bMag2RemoteClampRS;
	tyP0931MagConv2.tyCom.tyBtnRemoteUnclampRS.bValue		:= p_tyDI.bMag2RemoteUnclampRS;

	tyP0931MagConv2.tyCom.tyBtnSelUnclampRS.bValue			:= p_tyDI.bMag2SelUnClampRS;

	tyP0931MagConv2.tyCom.tyBtnCAB717Sen.bValue				:= p_tyDI.bMagConvCAB717MagSen2;
	tyP0931MagConv2.tyCom.tyBtnHeightSen.bValue				:= p_tyDI.bMagConvHeightSen2 OR p_tyDI.bHighMagDetSen2;
	tyP0931MagConv2.tyCom.tyBtnMagSmallSen.bValue			:= p_tyDI.bMagConvSmallMagSen2;
	tyP0931MagConv2.tyCom.tyBtnMagLargeSen.bValue			:= p_tyDI.bMagConvLargeMagSen2;
	tyP0931MagConv2.tyCom.tyBtnMagDetSen.bValue				:= p_tyDI.bMag2FixedSideDetect;
	tyP0931MagConv2.tyCom.tyBtnSltLckSen.bValue				:= p_tyDI.bSlotLckSenMag2;

	//Machine Bitmap //20
	IF p_tyNtParamCurr.eProjMag = LDMagDual AND p_tyNtParamCurr.bMagAutoVerifyPrep = FALSE THEN
		IF tyP0931MagConv2.tyFB.tyBtnFixedClamp.bRtCompl
			OR tyP0931MagConv2.tyDC.tyBtnFixedClamp.bRtCompl THEN

			tyP0931MagConv2.tyCom.tyBitmapMc.uiValueIdx	:= 44;

		ELSIF tyP0931MagConv2.tyFB.tyBtnFixedUnclamp.bRtCompl
			OR tyP0931MagConv2.tyDC.tyBtnFixedUnclamp.bRtCompl THEN

			tyP0931MagConv2.tyCom.tyBitmapMc.uiValueIdx	:= 43;

		ELSIF tyP0931MagConv2.tyFB.tyBtnRemoteClamp.bRtCompl
			OR tyP0931MagConv2.tyDC.tyBtnRemoteClamp.bRtCompl THEN

			tyP0931MagConv2.tyCom.tyBitmapMc.uiValueIdx	:= 49;

		ELSIF tyP0931MagConv2.tyFB.tyBtnRemoteUnclamp.bRtCompl
			OR tyP0931MagConv2.tyDC.tyBtnRemoteUnclamp.bRtCompl THEN

			tyP0931MagConv2.tyCom.tyBitmapMc.uiValueIdx	:= 48;

		ELSIF tyP0931MagConv2.tyFB.tyBtnEnt.bRtCompl OR tyP0931MagConv2.tyFB.tyBtnExit.bRtCompl OR tyP0931MagConv2.tyFB.tyBtnStop.bRtCompl
			OR tyP0931MagConv2.tyDC.tyBtnMagIn.bRtCompl OR tyP0931MagConv2.tyDC.tyBtnMagOut.bRtCompl OR tyP0931MagConv2.tyDC.tyBtnStop.bRtCompl THEN

			tyP0931MagConv2.tyCom.tyBitmapMc.uiValueIdx	:= 42;

		END_IF

	ELSIF p_tyNtParamCurr.eProjMag = LDMagDual AND p_tyNtParamCurr.bMagAutoVerifyPrep THEN
		IF tyP0931MagConv2.tyFB.tyBtnFixedClamp.bRtCompl
			OR tyP0931MagConv2.tyDC.tyBtnFixedClamp.bRtCompl THEN

			tyP0931MagConv2.tyCom.tyBitmapMc.uiValueIdx	:= 2;

		ELSIF tyP0931MagConv2.tyFB.tyBtnFixedUnclamp.bRtCompl
			OR tyP0931MagConv2.tyDC.tyBtnFixedUnclamp.bRtCompl THEN

			tyP0931MagConv2.tyCom.tyBitmapMc.uiValueIdx	:= 1;

		ELSIF tyP0931MagConv2.tyFB.tyBtnRemoteClamp.bRtCompl
			OR tyP0931MagConv2.tyDC.tyBtnRemoteClamp.bRtCompl THEN

			tyP0931MagConv2.tyCom.tyBitmapMc.uiValueIdx	:= 19;

		ELSIF tyP0931MagConv2.tyFB.tyBtnRemoteUnclamp.bRtCompl
			OR tyP0931MagConv2.tyDC.tyBtnRemoteUnclamp.bRtCompl THEN

			tyP0931MagConv2.tyCom.tyBitmapMc.uiValueIdx	:= 18;

		ELSIF tyP0931MagConv2.tyFB.tyBtnSelClamp.bRtCompl
			OR tyP0931MagConv2.tyDC.tyBtnSelClamp.bRtCompl THEN

			tyP0931MagConv2.tyCom.tyBitmapMc.uiValueIdx	:= 15;

		ELSIF tyP0931MagConv2.tyFB.tyBtnSelUnclamp.bRtCompl
			OR tyP0931MagConv2.tyDC.tyBtnSelUnclamp.bRtCompl THEN

			tyP0931MagConv2.tyCom.tyBitmapMc.uiValueIdx	:= 14;

		ELSIF tyP0931MagConv2.tyFB.tyBtnEnt.bRtCompl OR tyP0931MagConv2.tyFB.tyBtnExit.bRtCompl OR tyP0931MagConv2.tyFB.tyBtnStop.bRtCompl
			OR tyP0931MagConv2.tyDC.tyBtnMagIn.bRtCompl OR tyP0931MagConv2.tyDC.tyBtnMagOut.bRtCompl OR tyP0931MagConv2.tyDC.tyBtnStop.bRtCompl THEN

			tyP0931MagConv2.tyCom.tyBitmapMc.uiValueIdx	:= 0;

		END_IF
	ELSIF p_tyNtParamCurr.eProjMag = LDMagTriple AND p_tyNtParamCurr.bProjCurtainSenPrep = FALSE AND p_tyNtParamCurr.eCustomerReq <> Siemens AND p_tyNtParamCurr.eCustomerReq <> We_Fabricate THEN
		IF tyP0931MagConv2.tyFB.tyBtnFixedClamp.bRtCompl
			OR tyP0931MagConv2.tyDC.tyBtnFixedClamp.bRtCompl THEN

			tyP0931MagConv2.tyCom.tyBitmapMc.uiValueIdx	:= 2;

		ELSIF tyP0931MagConv2.tyFB.tyBtnFixedUnclamp.bRtCompl
			OR tyP0931MagConv2.tyDC.tyBtnFixedUnclamp.bRtCompl THEN

			tyP0931MagConv2.tyCom.tyBitmapMc.uiValueIdx	:= 1;

		ELSIF tyP0931MagConv2.tyFB.tyBtnRemoteClamp.bRtCompl
			OR tyP0931MagConv2.tyDC.tyBtnRemoteClamp.bRtCompl THEN

			tyP0931MagConv2.tyCom.tyBitmapMc.uiValueIdx	:= 15;

		ELSIF tyP0931MagConv2.tyFB.tyBtnRemoteUnclamp.bRtCompl
			OR tyP0931MagConv2.tyDC.tyBtnRemoteUnclamp.bRtCompl THEN

			tyP0931MagConv2.tyCom.tyBitmapMc.uiValueIdx	:= 14;

		ELSIF tyP0931MagConv2.tyFB.tyBtnSelClamp.bRtCompl
			OR tyP0931MagConv2.tyDC.tyBtnSelClamp.bRtCompl THEN

			tyP0931MagConv2.tyCom.tyBitmapMc.uiValueIdx	:= 21;

		ELSIF tyP0931MagConv2.tyFB.tyBtnSelUnclamp.bRtCompl
			OR tyP0931MagConv2.tyDC.tyBtnSelUnclamp.bRtCompl THEN

			tyP0931MagConv2.tyCom.tyBitmapMc.uiValueIdx	:= 20;

		ELSIF tyP0931MagConv2.tyFB.tyBtnEnt.bRtCompl OR tyP0931MagConv2.tyFB.tyBtnExit.bRtCompl OR tyP0931MagConv2.tyFB.tyBtnStop.bRtCompl
			OR tyP0931MagConv2.tyDC.tyBtnMagIn.bRtCompl OR tyP0931MagConv2.tyDC.tyBtnMagOut.bRtCompl OR tyP0931MagConv2.tyDC.tyBtnStop.bRtCompl THEN

			tyP0931MagConv2.tyCom.tyBitmapMc.uiValueIdx	:= 0;

		END_IF
	ELSIF p_tyNtParamCurr.eProjMag = LDMagTriple AND p_tyNtParamCurr.bProjCurtainSenPrep OR p_tyNtParamCurr.eCustomerReq = Siemens OR p_tyNtParamCurr.eCustomerReq = We_Fabricate THEN
		tyP0931MagConv2.tyCom.tyBitmapMc.uiValueIdx	:= 385-20;

	ELSIF p_tyNtParamCurr.eProjMag = LDMagQuadruple AND p_tyNtParamCurr.bMagAutoVerifyPrep THEN
		IF tyP0931MagConv2.tyFB.tyBtnFixedClamp.bRtCompl
			OR tyP0931MagConv2.tyDC.tyBtnFixedClamp.bRtCompl THEN

			tyP0931MagConv2.tyCom.tyBitmapMc.uiValueIdx	:= 72;

		ELSIF tyP0931MagConv2.tyFB.tyBtnFixedUnclamp.bRtCompl
			OR tyP0931MagConv2.tyDC.tyBtnFixedUnclamp.bRtCompl THEN

			tyP0931MagConv2.tyCom.tyBitmapMc.uiValueIdx	:= 71;

		ELSIF tyP0931MagConv2.tyFB.tyBtnRemoteClamp.bRtCompl
			OR tyP0931MagConv2.tyDC.tyBtnRemoteClamp.bRtCompl THEN

			tyP0931MagConv2.tyCom.tyBitmapMc.uiValueIdx	:= 74;

		ELSIF tyP0931MagConv2.tyFB.tyBtnRemoteUnclamp.bRtCompl
			OR tyP0931MagConv2.tyDC.tyBtnRemoteUnclamp.bRtCompl THEN

			tyP0931MagConv2.tyCom.tyBitmapMc.uiValueIdx	:= 73;

		ELSIF tyP0931MagConv2.tyFB.tyBtnSelClamp.bRtCompl
			OR tyP0931MagConv2.tyDC.tyBtnSelClamp.bRtCompl THEN

			tyP0931MagConv2.tyCom.tyBitmapMc.uiValueIdx	:= 76;

		ELSIF tyP0931MagConv2.tyFB.tyBtnSelUnclamp.bRtCompl
			OR tyP0931MagConv2.tyDC.tyBtnSelUnclamp.bRtCompl THEN

			tyP0931MagConv2.tyCom.tyBitmapMc.uiValueIdx	:= 75;

		ELSIF tyP0931MagConv2.tyFB.tyBtnEnt.bRtCompl OR tyP0931MagConv2.tyFB.tyBtnExit.bRtCompl OR tyP0931MagConv2.tyFB.tyBtnStop.bRtCompl
			OR tyP0931MagConv2.tyDC.tyBtnMagIn.bRtCompl OR tyP0931MagConv2.tyDC.tyBtnMagOut.bRtCompl OR tyP0931MagConv2.tyDC.tyBtnStop.bRtCompl THEN

			tyP0931MagConv2.tyCom.tyBitmapMc.uiValueIdx	:= 70;

		END_IF
	END_IF

	IF p_tyNtParamCurr.eProjMag = LDMagDual AND p_tyNtParamCurr.bMagAutoVerifyPrep = FALSE THEN
		IF tyP0931MagConv2.tyCom.tyBitmapMc.uiValueIdx < 100 THEN
			IF p_tyNtParamCurr.sJobNo = '2023-0276A01' THEN // no longer belt type //20 base
				tyP0931MagConv2.tyCom.tyBitmapMc.uiValueIdx	:= 494-20;
			ELSIF p_tyNtParamCurr.sJobNo = '2023-0258A01' THEN
				tyP0931MagConv2.tyCom.tyBitmapMc.uiValueIdx	:= 464-20;
			ELSE
				tyP0931MagConv2.tyCom.tyBitmapMc.uiValueIdx	:= tyP0931MagConv2.tyCom.tyBitmapMc.uiValueIdx + 100;
			END_IF
		END_IF
	ELSIF p_tyNtParamCurr.eProjMag = LDMagTriple AND p_tyNtParamCurr.bMagAutoVerifyPrep = FALSE AND p_tyNtParamCurr.bProjMotorizedPullerPrep = FALSE THEN
		IF tyP0931MagConv2.tyCom.tyBitmapMc.uiValueIdx < 100 THEN
			tyP0931MagConv2.tyCom.tyBitmapMc.uiValueIdx	:= tyP0931MagConv2.tyCom.tyBitmapMc.uiValueIdx + 100;
		END_IF
	ELSIF p_tyNtParamCurr.eProjMag = LDMagDual AND p_tyNtParamCurr.bMagAutoVerifyPrep = TRUE THEN
		IF tyP0931MagConv2.tyCom.tyBitmapMc.uiValueIdx < 200 THEN
			tyP0931MagConv2.tyCom.tyBitmapMc.uiValueIdx	:= tyP0931MagConv2.tyCom.tyBitmapMc.uiValueIdx + 200;
		END_IF
	ELSIF p_tyNtParamCurr.eProjMag = LDMagTriple AND p_tyNtParamCurr.bMagAutoVerifyPrep = FALSE AND p_tyNtParamCurr.bProjMotorizedPullerPrep = TRUE THEN
		IF tyP0931MagConv2.tyCom.tyBitmapMc.uiValueIdx < 300 THEN
			tyP0931MagConv2.tyCom.tyBitmapMc.uiValueIdx	:= tyP0931MagConv2.tyCom.tyBitmapMc.uiValueIdx + 300;
		END_IF
	END_IF

END_ACTION
```

#### Act_OptP0931Navi.st
```iecst
ACTION Act_OptP0931Navi:

	CASE p_tyNtParamCurr.eProjMag OF
		LDMagDual:
			IF tyP0931MagConv2.tyNavi2Lyr2.tyBtnBack.bRtCompl = TRUE THEN
				tyP0931MagConv2.tyNavi2Lyr2.tyBtnBack.bRtCompl	:= FALSE;
				tyP0931MagConv2.tyNavi2Lyr2.tyBtnBack.bValue	:= FALSE;

				eChgPage	:= UIP0920MtrNPneuCtrl;

				bDispMagConv1	:= FALSE;
				bDispMagConv2	:= TRUE;
				bDispMagConv3	:= FALSE;
				bDispMagConv4	:= FALSE;

			ELSIF tyP0931MagConv2.tyNavi2Lyr2.tyBtnLeft.bRtCompl = TRUE
				OR tyP0931MagConv2.tyNavi2Lyr2.tyBtnRgt.bRtCompl = TRUE
				THEN
				tyP0931MagConv2.tyNavi2Lyr2.tyBtnLeft.bRtCompl			:= FALSE;
				tyP0931MagConv2.tyNavi2Lyr2.tyBtnLeft.bValue			:= FALSE;
				tyP0931MagConv2.tyNavi2Lyr2.tyBtnRgt.bRtCompl			:= FALSE;
				tyP0931MagConv2.tyNavi2Lyr2.tyBtnRgt.bValue				:= FALSE;
				eChgPage												:= UIP0930MagConv1;
				bDispMagConv1	:= TRUE;
				bDispMagConv2	:= FALSE;
				bDispMagConv3	:= FALSE;
				bDispMagConv4	:= FALSE;
			END_IF

		LDMagTriple:
			IF tyP0931MagConv2.tyNavi3Lyr2.tyBtnBack.bRtCompl = TRUE THEN
				tyP0931MagConv2.tyNavi3Lyr2.tyBtnBack.bRtCompl	:= FALSE;
				tyP0931MagConv2.tyNavi3Lyr2.tyBtnBack.bValue	:= FALSE;

				eChgPage	:= UIP0920MtrNPneuCtrl;

				bDispMagConv1	:= FALSE;
				bDispMagConv2	:= TRUE;
				bDispMagConv3	:= FALSE;
				bDispMagConv4	:= FALSE;

			ELSIF tyP0931MagConv2.tyNavi3Lyr2.tyBtnLeft.bRtCompl = TRUE THEN
				tyP0931MagConv2.tyNavi3Lyr2.tyBtnLeft.bRtCompl			:= FALSE;
				tyP0931MagConv2.tyNavi3Lyr2.tyBtnLeft.bValue			:= FALSE;
				eChgPage												:= UIP0930MagConv1;

				bDispMagConv1	:= TRUE;
				bDispMagConv2	:= FALSE;
				bDispMagConv3	:= FALSE;
				bDispMagConv4	:= FALSE;

			ELSIF tyP0931MagConv2.tyNavi3Lyr2.tyBtnRgt.bRtCompl = TRUE THEN
				tyP0931MagConv2.tyNavi3Lyr2.tyBtnRgt.bRtCompl			:= FALSE;
				tyP0931MagConv2.tyNavi3Lyr2.tyBtnRgt.bValue				:= FALSE;
				eChgPage												:= UIP0932MagConv3;

				bDispMagConv1	:= FALSE;
				bDispMagConv2	:= FALSE;
				bDispMagConv3	:= TRUE;
				bDispMagConv4	:= FALSE;
			END_IF

		LDMagQuadruple:
			IF tyP0931MagConv2.tyNavi4Lyr2.tyBtnBack.bRtCompl = TRUE THEN
				tyP0931MagConv2.tyNavi4Lyr2.tyBtnBack.bRtCompl	:= FALSE;
				tyP0931MagConv2.tyNavi4Lyr2.tyBtnBack.bValue	:= FALSE;

				eChgPage	:= UIP0920MtrNPneuCtrl;
				bDispMagConv1	:= FALSE;
				bDispMagConv2	:= TRUE;
				bDispMagConv3	:= FALSE;
				bDispMagConv4	:= FALSE;

			ELSIF tyP0931MagConv2.tyNavi4Lyr2.tyBtnLeft.bRtCompl = TRUE THEN
				tyP0931MagConv2.tyNavi4Lyr2.tyBtnLeft.bRtCompl			:= FALSE;
				tyP0931MagConv2.tyNavi4Lyr2.tyBtnLeft.bValue			:= FALSE;
				eChgPage												:= UIP0930MagConv1;
				bDispMagConv1	:= TRUE;
				bDispMagConv2	:= FALSE;
				bDispMagConv3	:= FALSE;
				bDispMagConv4	:= FALSE;

			ELSIF tyP0931MagConv2.tyNavi4Lyr2.tyBtnRgt.bRtCompl = TRUE THEN
				tyP0931MagConv2.tyNavi4Lyr2.tyBtnRgt.bRtCompl			:= FALSE;
				tyP0931MagConv2.tyNavi4Lyr2.tyBtnRgt.bValue				:= FALSE;
				eChgPage												:= UIP0932MagConv3;
				bDispMagConv1	:= FALSE;
				bDispMagConv2	:= FALSE;
				bDispMagConv3	:= TRUE;
				bDispMagConv4	:= FALSE;
			END_IF
	END_CASE

END_ACTION
```

#### Act_OptP0931RstMnl.st
```iecst
ACTION Act_OptP0931RstMnl:

	IF EDGEPOS((bManualMod = FALSE) OR (p_eMagConv2Clp2Status = Error)) THEN

		eMagConv2Clp2Act	:= MagConv2ClpActIdle;
		eMagConvSelClp2Act	:= PneuActIdle;
		//Magazine Conveyor
		//FB
		tyP0931MagConv2.tyFB.tyBtnEnt.bRtCompl				:= FALSE;
		tyP0931MagConv2.tyFB.tyBtnExit.bRtCompl				:= FALSE;
		tyP0931MagConv2.tyFB.tyBtnStop.bRtCompl				:= FALSE;

		tyP0931MagConv2.tyFB.tyBtnEnt.bValue				:= FALSE;
		tyP0931MagConv2.tyFB.tyBtnExit.bValue				:= FALSE;
		tyP0931MagConv2.tyFB.tyBtnStop.bValue				:= TRUE;

		tyP0931MagConv2.tyFB.tyBtnEnt.bRtLk					:= FALSE;
		tyP0931MagConv2.tyFB.tyBtnExit.bRtLk				:= FALSE;
		tyP0931MagConv2.tyFB.tyBtnStop.bRtLk				:= TRUE;

		tyP0931MagConv2.tyFB.tyBtnEnt.uiMaskRtStat.0		:= TRUE;
		tyP0931MagConv2.tyFB.tyBtnExit.uiMaskRtStat.0		:= TRUE;
		tyP0931MagConv2.tyCom.tyBtnSwitch.uiMaskRtStat.0	:= TRUE;

		//Direct
		tyP0931MagConv2.tyDC.tyBtnMagIn.bRtCompl			:= FALSE;
		tyP0931MagConv2.tyDC.tyBtnMagOut.bRtCompl			:= FALSE;
		tyP0931MagConv2.tyDC.tyBtnStop.bRtCompl				:= FALSE;

		tyP0931MagConv2.tyDC.tyBtnMagIn.bValue				:= FALSE;
		tyP0931MagConv2.tyDC.tyBtnMagOut.bValue				:= FALSE;
		tyP0931MagConv2.tyDC.tyBtnStop.bValue				:= TRUE;

		tyP0931MagConv2.tyDC.tyBtnMagIn.bRtLk				:= FALSE;
		tyP0931MagConv2.tyDC.tyBtnMagOut.bRtLk				:= FALSE;
		tyP0931MagConv2.tyDC.tyBtnStop.bRtLk				:= TRUE;

		tyP0931MagConv2.tyDC.tyBtnMagIn.uiMaskRtStat.0		:= TRUE;
		tyP0931MagConv2.tyDC.tyBtnMagOut.uiMaskRtStat.0		:= TRUE;
		tyP0931MagConv2.tyCom.tyBtnSwitch.uiMaskRtStat.0	:= TRUE;

		//Magazine Clamper
		//FB
		//Fixed/Bottom
		tyP0931MagConv2.tyFB.tyBtnFixedClamp.bRtCompl			:= FALSE;
		tyP0931MagConv2.tyFB.tyBtnFixedUnclamp.bRtCompl			:= FALSE;

		tyP0931MagConv2.tyFB.tyBtnFixedClamp.bValue				:= FALSE;
		tyP0931MagConv2.tyFB.tyBtnFixedUnclamp.bValue			:= FALSE;

		//Remote/Top
		tyP0931MagConv2.tyFB.tyBtnRemoteClamp.bRtCompl			:= FALSE;
		tyP0931MagConv2.tyFB.tyBtnRemoteUnclamp.bRtCompl		:= FALSE;

		tyP0931MagConv2.tyFB.tyBtnRemoteClamp.bValue			:= FALSE;
		tyP0931MagConv2.tyFB.tyBtnRemoteUnclamp.bValue			:= FALSE;

		//Selection
		tyP0931MagConv2.tyFB.tyBtnSelClamp.bRtCompl			:= FALSE;
		tyP0931MagConv2.tyFB.tyBtnSelUnclamp.bRtCompl		:= FALSE;

		tyP0931MagConv2.tyFB.tyBtnSelClamp.bValue			:= FALSE;
		tyP0931MagConv2.tyFB.tyBtnSelUnclamp.bValue			:= FALSE;

		tyP0931MagConv2.tyFB.tyBtnFixedClamp.uiMaskRtStat.0		:= TRUE;
		tyP0931MagConv2.tyFB.tyBtnFixedUnclamp.uiMaskRtStat.0	:= TRUE;
		tyP0931MagConv2.tyFB.tyBtnRemoteClamp.uiMaskRtStat.0	:= TRUE;
		tyP0931MagConv2.tyFB.tyBtnRemoteUnclamp.uiMaskRtStat.0	:= TRUE;
		tyP0931MagConv2.tyFB.tyBtnSelClamp.uiMaskRtStat.0		:= TRUE;
		tyP0931MagConv2.tyFB.tyBtnSelUnclamp.uiMaskRtStat.0		:= TRUE;

		tyP0931MagConv2.tyCom.tyBtnSwitch.uiMaskRtStat.0		:= TRUE;

		//Direct
		//Fixed/Bottom
		tyP0931MagConv2.tyDC.tyBtnFixedClamp.bRtCompl			:= FALSE;
		tyP0931MagConv2.tyDC.tyBtnFixedUnclamp.bRtCompl			:= FALSE;

		tyP0931MagConv2.tyDC.tyBtnFixedClamp.bValue				:= FALSE;
		tyP0931MagConv2.tyDC.tyBtnFixedUnclamp.bValue			:= FALSE;

		//Remote/Top
		tyP0931MagConv2.tyDC.tyBtnRemoteClamp.bRtCompl			:= FALSE;
		tyP0931MagConv2.tyDC.tyBtnRemoteUnclamp.bRtCompl		:= FALSE;

		tyP0931MagConv2.tyDC.tyBtnRemoteClamp.bValue			:= FALSE;
		tyP0931MagConv2.tyDC.tyBtnRemoteUnclamp.bValue			:= FALSE;

		//Selection
		tyP0931MagConv2.tyDC.tyBtnSelClamp.bRtCompl				:= FALSE;
		tyP0931MagConv2.tyDC.tyBtnSelUnclamp.bRtCompl			:= FALSE;

		tyP0931MagConv2.tyDC.tyBtnSelClamp.bValue				:= FALSE;
		tyP0931MagConv2.tyDC.tyBtnSelUnclamp.bValue				:= FALSE;

		tyP0931MagConv2.tyDC.tyBtnFixedClamp.uiMaskRtStat.0		:= TRUE;
		tyP0931MagConv2.tyDC.tyBtnFixedUnclamp.uiMaskRtStat.0	:= TRUE;
		tyP0931MagConv2.tyDC.tyBtnRemoteClamp.uiMaskRtStat.0	:= TRUE;
		tyP0931MagConv2.tyDC.tyBtnRemoteUnclamp.uiMaskRtStat.0	:= TRUE;
		tyP0931MagConv2.tyDC.tyBtnSelClamp.uiMaskRtStat.0		:= TRUE;
		tyP0931MagConv2.tyDC.tyBtnSelUnclamp.uiMaskRtStat.0		:= TRUE;

		tyP0931MagConv2.tyCom.tyBtnSwitch.uiMaskRtStat.0		:= TRUE;

	END_IF

	IF EDGEPOS(bManualMod = FALSE) THEN
		tyP0931MagConv2.tyCom.tyBtnSwitch.bValue := FALSE;

		IF p_tyNtParamCurr.bMagAutoVerifyPrep = FALSE THEN
			fUIInRtStatHide(ADR(tyP0931MagConv2.tyDC.tyLyrWithoutSelClamp.uiRtStat));
			fUIInRtStatOff(ADR(tyP0931MagConv2.tyFB.tyLyrWithoutSelClamp.uiRtStat));
		ELSE

			fUIInRtStatHide(ADR(tyP0931MagConv2.tyDC.tyLyr.uiRtStat));
			fUIInRtStatOff(ADR(tyP0931MagConv2.tyFB.tyLyr.uiRtStat));
		END_IF
	END_IF
END_ACTION
```

#### Act_EntP0932Disp.st
```iecst
ACTION Act_EntP0932Disp:

	//Access Address
	p_tyC0002FullMask ACCESS ADR(tyP0932MagConv3.tyFullMaskHide);

//	p_tyC0004Navi ACCESS ADR(tyP0932MagConv3.tyNaviBack);
	CASE p_tyNtParamCurr.eProjMag OF
		LDMagTriple:
			p_tyC0004Navi ACCESS ADR(tyP0932MagConv3.tyNavi3Lyr3);
		LDMagQuadruple:
			p_tyC0004Navi ACCESS ADR(tyP0932MagConv3.tyNavi4Lyr3);
	END_CASE

	p_tyC0005Main ACCESS ADR(tyCommon.tyMain);

	p_tyC0007Notif ACCESS ADR(tyCommon.tyNotif);

	p_tyC0008MsgBox ACCESS ADR(tyP0932MagConv3.tyMsgBoxHide);

	p_tyC0009Info ACCESS ADR(tyCommon.tyInfo);

	p_tyP0932Mag3ConvCom ACCESS ADR(tyP0932MagConv3.tyCom);
	p_tyP0932Mag3ConvDC ACCESS ADR(tyP0932MagConv3.tyDC);
	p_tyP0932Mag3ConvFB ACCESS ADR(tyP0932MagConv3.tyFB);

	IF p_tyNtParamCurr.eProjMag = LDMagDual AND p_tyNtParamCurr.bMagAutoVerifyPrep = FALSE THEN
		tyP0932MagConv3.tyCom.tyBitmapMc.usiValueIdx	:= 111;
	ELSIF p_tyNtParamCurr.eProjMag = LDMagDual AND p_tyNtParamCurr.bMagAutoVerifyPrep = TRUE THEN
		tyP0932MagConv3.tyCom.tyBitmapMc.usiValueIdx	:= 200;
	ELSIF p_tyNtParamCurr.eProjMag = LDMagTriple AND p_tyNtParamCurr.bMagAutoVerifyPrep = TRUE THEN
		tyP0932MagConv3.tyCom.tyBitmapMc.usiValueIdx	:= 0;
	ELSIF p_tyNtParamCurr.eProjMag = LDMagQuadruple AND p_tyNtParamCurr.bMagAutoVerifyPrep = TRUE THEN
		tyP0932MagConv3.tyCom.tyBitmapMc.usiValueIdx	:= 109;
	ELSE
		tyP0932MagConv3.tyCom.tyBitmapMc.usiValueIdx	:= 100;
	END_IF

	IF p_tyNtParamCurr.bMagAutoVerifyPrep = FALSE THEN
		tyP0932MagConv3.tyFB.tyBtnFixedClamp.usiTxtIdx	:= 6;
		tyP0932MagConv3.tyFB.tyBtnFixedUnclamp.usiTxtIdx:= 6;
		tyP0932MagConv3.tyFB.tyBtnRemoteClamp.usiTxtIdx	:= 6;
		tyP0932MagConv3.tyFB.tyBtnRemoteUnclamp.usiTxtIdx:= 6;
	ELSE
		tyP0932MagConv3.tyFB.tyBtnFixedClamp.usiTxtIdx	:= 6;
		tyP0932MagConv3.tyFB.tyBtnFixedUnclamp.usiTxtIdx:= 6;
		tyP0932MagConv3.tyFB.tyBtnRemoteClamp.usiTxtIdx	:= 6;
		tyP0932MagConv3.tyFB.tyBtnRemoteUnclamp.usiTxtIdx:= 6;

	END_IF

	IF p_tyNtParamCurr.bMagAutoVerifyPrep = FALSE THEN
		IF tyP0932MagConv3.tyCom.tyBtnSwitch.bValue THEN
			fUIInRtStatHide(ADR(tyP0932MagConv3.tyFB.tyLyr.uiRtStat));
			fUIInRtStatHide(ADR(tyP0932MagConv3.tyDC.tyLyr.uiRtStat));
			fUIInRtStatHide(ADR(tyP0932MagConv3.tyFB.tyLyrWithoutSelClamp.uiRtStat));
			fUIInRtStatOff(ADR(tyP0932MagConv3.tyDC.tyLyrWithoutSelClamp.uiRtStat));
		ELSE
			fUIInRtStatHide(ADR(tyP0932MagConv3.tyFB.tyLyr.uiRtStat));
			fUIInRtStatHide(ADR(tyP0932MagConv3.tyDC.tyLyr.uiRtStat));
			fUIInRtStatOff(ADR(tyP0932MagConv3.tyFB.tyLyrWithoutSelClamp.uiRtStat));
			fUIInRtStatHide(ADR(tyP0932MagConv3.tyDC.tyLyrWithoutSelClamp.uiRtStat));
		END_IF
	ELSE
		IF tyP0932MagConv3.tyCom.tyBtnSwitch.bValue THEN
			fUIInRtStatHide(ADR(tyP0932MagConv3.tyFB.tyLyr.uiRtStat));
			fUIInRtStatOff(ADR(tyP0932MagConv3.tyDC.tyLyr.uiRtStat));
			fUIInRtStatHide(ADR(tyP0932MagConv3.tyFB.tyLyrWithoutSelClamp.uiRtStat));
			fUIInRtStatHide(ADR(tyP0932MagConv3.tyDC.tyLyrWithoutSelClamp.uiRtStat));
		ELSE
			fUIInRtStatOff(ADR(tyP0932MagConv3.tyFB.tyLyr.uiRtStat));
			fUIInRtStatHide(ADR(tyP0932MagConv3.tyDC.tyLyr.uiRtStat));
			fUIInRtStatHide(ADR(tyP0932MagConv3.tyFB.tyLyrWithoutSelClamp.uiRtStat));
			fUIInRtStatHide(ADR(tyP0932MagConv3.tyDC.tyLyrWithoutSelClamp.uiRtStat));
		END_IF
	END_IF

END_ACTION
```

#### Act_OptP0932FullMask.st
```iecst
ACTION Act_OptP0932FullMask:

	IF eCurrPage = UIP0932MagConv3 THEN

		IF p_tyDI.bEStopSig = FALSE THEN
			p_tyC0002FullMask ACCESS ADR(tyP0932MagConv3.tyFullMaskEStop);

		ELSIF p_tyDI.bCoverSWSig = FALSE THEN
			p_tyC0002FullMask ACCESS ADR(tyP0932MagConv3.tyFullMaskCWSig);

		ELSIF p_tyDI.bSafetyRlySig = FALSE THEN
			p_tyC0002FullMask ACCESS ADR(tyP0932MagConv3.tyFullMaskSafetyRly);

		ELSE
			p_tyC0002FullMask ACCESS ADR(tyP0932MagConv3.tyFullMaskHide);

		END_IF

	END_IF

END_ACTION
```

#### Act_OptP0932MagConv3ChgLyr.st
```iecst
ACTION Act_OptP0932MagConv3ChgLyr:

	IF p_tyNtParamCurr.bMagAutoVerifyPrep THEN
		IF tyP0932MagConv3.tyCom.tyBtnSwitch.bRtCompl THEN
			tyP0932MagConv3.tyCom.tyBtnSwitch.bRtCompl	:= FALSE;

			IF tyP0932MagConv3.tyCom.tyBtnSwitch.bValue = TRUE THEN
				fUIInRtStatOff(ADR(tyP0932MagConv3.tyDC.tyLyr.uiRtStat));
				fUIInRtStatHide(ADR(tyP0932MagConv3.tyFB.tyLyr.uiRtStat));
			ELSE
				fUIInRtStatHide(ADR(tyP0932MagConv3.tyDC.tyLyr.uiRtStat));
				fUIInRtStatOff(ADR(tyP0932MagConv3.tyFB.tyLyr.uiRtStat));
			END_IF

		END_IF
	ELSE
		IF tyP0932MagConv3.tyCom.tyBtnSwitch.bRtCompl THEN
			tyP0932MagConv3.tyCom.tyBtnSwitch.bRtCompl	:= FALSE;

			IF tyP0932MagConv3.tyCom.tyBtnSwitch.bValue = TRUE THEN
				fUIInRtStatOff(ADR(tyP0932MagConv3.tyDC.tyLyrWithoutSelClamp.uiRtStat));
				fUIInRtStatHide(ADR(tyP0932MagConv3.tyFB.tyLyrWithoutSelClamp.uiRtStat));
			ELSE
				fUIInRtStatHide(ADR(tyP0932MagConv3.tyDC.tyLyrWithoutSelClamp.uiRtStat));
				fUIInRtStatOff(ADR(tyP0932MagConv3.tyFB.tyLyrWithoutSelClamp.uiRtStat));
			END_IF

		END_IF
	END_IF

END_ACTION
```

#### Act_OptP0932MagConv3DC.st
```iecst
ACTION Act_OptP0932MagConv3DC:

	//Magazine Conveyor
	IF tyP0932MagConv3.tyDC.tyBtnStop.bRtCompl = TRUE THEN
		eMagConv2Clp3Act	:= MagConv2ClpActStop;

		IF p_eMagConv2Clp3Stat = MagConv2ClpActStop AND p_eMagConv2Clp3Status = Done THEN
			eMagConv2Clp3Act	:= MagConv2ClpActIdle;

			tyP0932MagConv3.tyDC.tyBtnStop.bRtCompl		:= FALSE;
			tyP0932MagConv3.tyDC.tyBtnStop.bValue		:= TRUE;
			tyP0932MagConv3.tyDC.tyBtnStop.bRtLk		:= TRUE;

			tyP0932MagConv3.tyDC.tyBtnMagIn.bRtCompl	:= FALSE;
			tyP0932MagConv3.tyDC.tyBtnMagIn.bValue		:= FALSE;
			tyP0932MagConv3.tyDC.tyBtnMagIn.bRtLk		:= FALSE;

			tyP0932MagConv3.tyDC.tyBtnMagOut.bRtCompl	:= FALSE;
			tyP0932MagConv3.tyDC.tyBtnMagOut.bValue		:= FALSE;
			tyP0932MagConv3.tyDC.tyBtnMagOut.bRtLk		:= FALSE;
		END_IF

	ELSIF tyP0932MagConv3.tyDC.tyBtnMagIn.bRtCompl = TRUE THEN
		tyP0932MagConv3.tyDC.tyBtnMagIn.bValue	:= TRUE;
		tyP0932MagConv3.tyDC.tyBtnMagIn.bRtLk	:= TRUE;

		tyP0932MagConv3.tyDC.tyBtnStop.bValue	:= FALSE;
		tyP0932MagConv3.tyDC.tyBtnStop.bRtLk	:= FALSE;

		IF p_tyNtParamCurr.eProjMagConvDir = ConvDirLToR OR p_tyNtParamCurr.eProjMagConvDir = ConvDirLToL THEN

			eMagConv2Clp3Act	:= MagConv2ClpActSetMtrSigOnOrLToR;

			IF p_eMagConv2Clp3Stat = MagConv2ClpActSetMtrSigOnOrLToR AND p_eMagConv2Clp3Status = Done THEN
				eMagConv2Clp3Act	:= MagConv2ClpActIdle;

				tyP0932MagConv3.tyDC.tyBtnMagIn.bRtCompl	:= FALSE;
			END_IF

		ELSE

			eMagConv2Clp3Act	:= MagConv2ClpActSetMtrDirOrRToL;

			IF p_eMagConv2Clp3Stat = MagConv2ClpActSetMtrDirOrRToL AND p_eMagConv2Clp3Status = Done THEN
				eMagConv2Clp3Act	:= MagConv2ClpActIdle;

				tyP0932MagConv3.tyDC.tyBtnMagIn.bRtCompl	:= FALSE;
			END_IF

		END_IF

	ELSIF tyP0932MagConv3.tyDC.tyBtnMagOut.bRtCompl = TRUE THEN
		tyP0932MagConv3.tyDC.tyBtnMagOut.bValue	:= TRUE;
		tyP0932MagConv3.tyDC.tyBtnMagOut.bRtLk	:= TRUE;

		tyP0932MagConv3.tyDC.tyBtnStop.bValue	:= FALSE;
		tyP0932MagConv3.tyDC.tyBtnStop.bRtLk	:= FALSE;

		IF p_tyNtParamCurr.eProjMagConvDir = ConvDirLToR OR p_tyNtParamCurr.eProjMagConvDir = ConvDirRToR THEN

			eMagConv2Clp3Act	:= MagConv2ClpActSetMtrSigOnOrLToR;

			IF p_eMagConv2Clp3Stat = MagConv2ClpActSetMtrSigOnOrLToR AND p_eMagConv2Clp3Status = Done THEN
				eMagConv2Clp3Act	:= MagConv2ClpActIdle;

				tyP0932MagConv3.tyDC.tyBtnMagOut.bRtCompl	:= FALSE;
			END_IF

		ELSE

			eMagConv2Clp3Act	:= MagConv2ClpActSetMtrDirOrRToL;

			IF p_eMagConv2Clp3Stat = MagConv2ClpActSetMtrDirOrRToL AND p_eMagConv2Clp3Status = Done THEN
				eMagConv2Clp3Act	:= MagConv2ClpActIdle;

				tyP0932MagConv3.tyDC.tyBtnMagOut.bRtCompl	:= FALSE;
			END_IF

		END_IF

	END_IF

	//Magazine Clamper
	IF tyP0932MagConv3.tyCom.tyBtnSwitch.bValue = TRUE THEN
		IF p_bSelClamp3TwoCtrlOut = FALSE THEN
			IF tyP0932MagConv3.tyDC.tyBtnSelUnclamp.bRtCompl = TRUE THEN
				tyP0932MagConv3.tyDC.tyBtnSelUnclamp.bValue := TRUE;
				tyP0932MagConv3.tyDC.tyBtnSelClamp.bValue := FALSE;

				eMagConvSelClp3Act	:= PneuActSetExt;

				IF p_eSelClamp3Stat = PneuActSetExt AND p_eSelClamp3Status = Done THEN
					eMagConvSelClp3Act	:= PneuActIdle;

					tyP0932MagConv3.tyDC.tyBtnSelUnclamp.bRtCompl	:= FALSE;
				END_IF

			ELSIF tyP0932MagConv3.tyDC.tyBtnSelClamp.bRtCompl = TRUE THEN
				tyP0932MagConv3.tyDC.tyBtnSelClamp.bValue := TRUE;
				tyP0932MagConv3.tyDC.tyBtnSelUnclamp.bValue := FALSE;

				eMagConvSelClp3Act	:= PneuActSetRet;

				IF p_eSelClamp3Stat = PneuActSetRet AND p_eSelClamp3Status = Done THEN
					eMagConvSelClp3Act	:= PneuActIdle;

					tyP0932MagConv3.tyDC.tyBtnSelClamp.bRtCompl	:= FALSE;
				END_IF
			END_IF

		ELSE
			IF (tyP0932MagConv3.tyDC.tyBtnSelUnclamp.bRtCompl = TRUE) OR (tyP0932MagConv3.tyDC.tyBtnSelClamp.bRtCompl = TRUE) THEN
				IF (tyP0932MagConv3.tyDC.tyBtnSelUnclamp.bValue = TRUE) AND (tyP0932MagConv3.tyDC.tyBtnSelClamp.bValue = TRUE) THEN
					eMagConvSelClp3Act	:= PneuActSetAll;

					IF p_eSelClamp3Stat = PneuActSetAll AND p_eSelClamp3Status = Done THEN
						eMagConvSelClp3Act	:= PneuActIdle;

						tyP0932MagConv3.tyDC.tyBtnSelUnclamp.bRtCompl		:= FALSE;
						tyP0932MagConv3.tyDC.tyBtnSelClamp.bRtCompl			:= FALSE;
					END_IF

				ELSIF (tyP0932MagConv3.tyDC.tyBtnSelUnclamp.bValue = TRUE) AND (tyP0932MagConv3.tyDC.tyBtnSelClamp.bValue = FALSE) THEN
					eMagConvSelClp3Act	:= PneuActSetExt;

					IF p_eSelClamp3Stat = PneuActSetExt AND p_eSelClamp3Status = Done THEN
						eMagConvSelClp3Act	:= PneuActIdle;

						tyP0932MagConv3.tyDC.tyBtnSelUnclamp.bRtCompl		:= FALSE;
						tyP0932MagConv3.tyDC.tyBtnSelClamp.bRtCompl			:= FALSE;
					END_IF

				ELSIF (tyP0932MagConv3.tyDC.tyBtnSelUnclamp.bValue = FALSE) AND (tyP0932MagConv3.tyDC.tyBtnSelClamp.bValue = TRUE) THEN
					eMagConvSelClp3Act	:= PneuActSetRet;

					IF p_eSelClamp3Stat = PneuActSetRet AND p_eSelClamp3Status = Done THEN
						eMagConvSelClp3Act	:= PneuActIdle;

						tyP0932MagConv3.tyDC.tyBtnSelUnclamp.bRtCompl		:= FALSE;
						tyP0932MagConv3.tyDC.tyBtnSelClamp.bRtCompl			:= FALSE;
					END_IF

				ELSE
					eMagConvSelClp3Act	:= PneuActRstAll;

					IF p_eSelClamp3Stat = PneuActRstAll AND p_eSelClamp3Status = Done THEN
						eMagConvSelClp3Act	:= PneuActIdle;

						tyP0932MagConv3.tyDC.tyBtnSelUnclamp.bRtCompl		:= FALSE;
						tyP0932MagConv3.tyDC.tyBtnSelClamp.bRtCompl			:= FALSE;
					END_IF

				END_IF
			END_IF
		END_IF
		IF p_bMagConv2Clp1ClprTwoOutputCtrl = FALSE THEN

			//Fixed
			IF tyP0932MagConv3.tyDC.tyBtnFixedClamp.bRtCompl = TRUE THEN
				tyP0932MagConv3.tyDC.tyBtnFixedClamp.bValue		:= TRUE;
				tyP0932MagConv3.tyDC.tyBtnFixedUnclamp.bValue	:= FALSE;

				eMagConv2Clp3Act	:= MagConv2ClpActFixClprSetClamp;

				IF p_eMagConv2Clp3Stat = MagConv2ClpActFixClprSetClamp AND p_eMagConv2Clp3Status = Done THEN
					eMagConv2Clp3Act	:= MagConv2ClpActIdle;

					tyP0932MagConv3.tyDC.tyBtnFixedClamp.bRtCompl	:= FALSE;
				END_IF

			ELSIF tyP0932MagConv3.tyDC.tyBtnFixedUnclamp.bRtCompl = TRUE THEN
				tyP0932MagConv3.tyDC.tyBtnFixedUnclamp.bValue	:= TRUE;
				tyP0932MagConv3.tyDC.tyBtnFixedClamp.bValue		:= FALSE;

				eMagConv2Clp3Act	:= MagConv2ClpActFixClprSetUnclamp;

				IF p_eMagConv2Clp3Stat = MagConv2ClpActFixClprSetUnclamp AND p_eMagConv2Clp3Status = Done THEN
					eMagConv2Clp3Act	:= MagConv2ClpActIdle;

					tyP0932MagConv3.tyDC.tyBtnFixedUnclamp.bRtCompl	:= FALSE;
				END_IF

			END_IF

			//Remote
			IF tyP0932MagConv3.tyDC.tyBtnRemoteClamp.bRtCompl = TRUE THEN
				tyP0932MagConv3.tyDC.tyBtnRemoteClamp.bValue		:= TRUE;
				tyP0932MagConv3.tyDC.tyBtnRemoteUnclamp.bValue		:= FALSE;

				eMagConv2Clp3Act	:= MagConv2ClpActRmtClprSetClamp;

				IF p_eMagConv2Clp3Stat = MagConv2ClpActRmtClprSetClamp AND p_eMagConv2Clp3Status = Done THEN
					eMagConv2Clp3Act	:= MagConv2ClpActIdle;

					tyP0932MagConv3.tyDC.tyBtnRemoteClamp.bRtCompl	:= FALSE;
				END_IF

			ELSIF tyP0932MagConv3.tyDC.tyBtnRemoteUnclamp.bRtCompl = TRUE THEN
				tyP0932MagConv3.tyDC.tyBtnRemoteUnclamp.bValue	:= TRUE;
				tyP0932MagConv3.tyDC.tyBtnRemoteClamp.bValue	:= FALSE;

				eMagConv2Clp3Act	:= MagConv2ClpActRmtClprSetUnclamp;

				IF p_eMagConv2Clp3Stat = MagConv2ClpActRmtClprSetUnclamp AND p_eMagConv2Clp3Status = Done THEN
					eMagConv2Clp3Act	:= MagConv2ClpActIdle;

					tyP0932MagConv3.tyDC.tyBtnRemoteUnclamp.bRtCompl	:= FALSE;
				END_IF

			END_IF

		ELSE

			//Fixed
			IF (tyP0932MagConv3.tyDC.tyBtnFixedClamp.bRtCompl = TRUE) OR (tyP0932MagConv3.tyDC.tyBtnFixedUnclamp.bRtCompl = TRUE) THEN

				IF (tyP0932MagConv3.tyDC.tyBtnFixedClamp.bValue = TRUE) AND (tyP0932MagConv3.tyDC.tyBtnFixedUnclamp.bValue = TRUE) THEN

					eMagConv2Clp3Act	:= MagConv2ClpActFixClprSetAll;

					IF p_eMagConv2Clp3Stat = MagConv2ClpActFixClprSetAll AND p_eMagConv2Clp3Status = Done THEN

						eMagConv2Clp3Act	:= MagConv2ClpActIdle;

						tyP0932MagConv3.tyDC.tyBtnFixedClamp.bRtCompl	:= FALSE;
						tyP0932MagConv3.tyDC.tyBtnFixedUnclamp.bRtCompl	:= FALSE;
					END_IF

				ELSIF (tyP0932MagConv3.tyDC.tyBtnFixedClamp.bValue = TRUE) AND (tyP0932MagConv3.tyDC.tyBtnFixedUnclamp.bValue = FALSE) THEN
					eMagConv2Clp3Act	:= MagConv2ClpActFixClprSetClamp;

					IF p_eMagConv2Clp3Stat = MagConv2ClpActFixClprSetClamp AND p_eMagConv2Clp3Status = Done THEN

						eMagConv2Clp3Act	:= MagConv2ClpActIdle;

						tyP0932MagConv3.tyDC.tyBtnFixedClamp.bRtCompl	:= FALSE;
						tyP0932MagConv3.tyDC.tyBtnFixedUnclamp.bRtCompl	:= FALSE;
					END_IF

				ELSIF (tyP0932MagConv3.tyDC.tyBtnFixedClamp.bValue = FALSE) AND (tyP0932MagConv3.tyDC.tyBtnFixedUnclamp.bValue = TRUE) THEN
					eMagConv2Clp3Act	:= MagConv2ClpActFixClprSetUnclamp;

					IF p_eMagConv2Clp3Stat = MagConv2ClpActFixClprSetUnclamp AND p_eMagConv2Clp3Status = Done THEN

						eMagConv2Clp3Act	:= MagConv2ClpActIdle;

						tyP0932MagConv3.tyDC.tyBtnFixedClamp.bRtCompl	:= FALSE;
						tyP0932MagConv3.tyDC.tyBtnFixedUnclamp.bRtCompl	:= FALSE;
					END_IF

				ELSE
					eMagConv2Clp3Act	:= MagConv2ClpActFixClprRstAll;

					IF p_eMagConv2Clp3Stat = MagConv2ClpActFixClprRstAll AND p_eMagConv2Clp3Status = Done THEN

						eMagConv2Clp3Act	:= MagConv2ClpActIdle;

						tyP0932MagConv3.tyDC.tyBtnFixedClamp.bRtCompl	:= FALSE;
						tyP0932MagConv3.tyDC.tyBtnFixedUnclamp.bRtCompl	:= FALSE;
					END_IF

				END_IF

				//Remote
				IF (tyP0932MagConv3.tyDC.tyBtnRemoteClamp.bRtCompl = TRUE) OR (tyP0932MagConv3.tyDC.tyBtnRemoteUnclamp.bRtCompl = TRUE) THEN

					IF (tyP0932MagConv3.tyDC.tyBtnRemoteClamp.bValue = TRUE) AND (tyP0932MagConv3.tyDC.tyBtnRemoteUnclamp.bValue = TRUE) THEN

						eMagConv2Clp3Act	:= MagConv2ClpActRmtClprSetAll;

						IF p_eMagConv2Clp3Stat = MagConv2ClpActRmtClprSetAll AND p_eMagConv2Clp3Status = Done THEN

							eMagConv2Clp3Act	:= MagConv2ClpActIdle;

							tyP0932MagConv3.tyDC.tyBtnRemoteClamp.bRtCompl		:= FALSE;
							tyP0932MagConv3.tyDC.tyBtnRemoteUnclamp.bRtCompl	:= FALSE;
						END_IF

					ELSIF (tyP0932MagConv3.tyDC.tyBtnRemoteClamp.bValue = TRUE) AND (tyP0932MagConv3.tyDC.tyBtnRemoteUnclamp.bValue = FALSE) THEN
						eMagConv2Clp3Act	:= MagConv2ClpActRmtClprSetClamp;

						IF p_eMagConv2Clp3Stat = MagConv2ClpActRmtClprSetClamp AND p_eMagConv2Clp3Status = Done THEN

							eMagConv2Clp3Act	:= MagConv2ClpActIdle;

							tyP0932MagConv3.tyDC.tyBtnRemoteClamp.bRtCompl	:= FALSE;
							tyP0932MagConv3.tyDC.tyBtnRemoteUnclamp.bRtCompl	:= FALSE;
						END_IF

					ELSIF (tyP0932MagConv3.tyDC.tyBtnRemoteClamp.bValue = FALSE) AND (tyP0932MagConv3.tyDC.tyBtnRemoteUnclamp.bValue = TRUE) THEN
						eMagConv2Clp3Act	:= MagConv2ClpActRmtClprSetUnclamp;

						IF p_eMagConv2Clp3Stat = MagConv2ClpActRmtClprSetUnclamp AND p_eMagConv2Clp3Status = Done THEN

							eMagConv2Clp3Act	:= MagConv2ClpActIdle;

							tyP0932MagConv3.tyDC.tyBtnRemoteClamp.bRtCompl	:= FALSE;
							tyP0932MagConv3.tyDC.tyBtnRemoteUnclamp.bRtCompl	:= FALSE;
						END_IF

					ELSE
						eMagConv2Clp3Act	:= MagConv2ClpActRmtClprRstAll;

						IF p_eMagConv2Clp3Stat = MagConv2ClpActRmtClprRstAll AND p_eMagConv2Clp3Status = Done THEN

							eMagConv2Clp3Act	:= MagConv2ClpActIdle;

							tyP0932MagConv3.tyDC.tyBtnRemoteClamp.bRtCompl	:= FALSE;
							tyP0932MagConv3.tyDC.tyBtnRemoteUnclamp.bRtCompl	:= FALSE;
						END_IF

					END_IF
				END_IF

			END_IF

		END_IF

		//Fixed
		tyP0932MagConv3.tyFB.tyBtnFixedClamp.bRtCompl		:= FALSE;
		tyP0932MagConv3.tyFB.tyBtnFixedClamp.bValue			:= FALSE;
		tyP0932MagConv3.tyFB.tyBtnFixedUnclamp.bRtCompl		:= FALSE;
		tyP0932MagConv3.tyFB.tyBtnFixedUnclamp.bValue		:= FALSE;

		//Remote
		tyP0932MagConv3.tyFB.tyBtnRemoteClamp.bRtCompl		:= FALSE;
		tyP0932MagConv3.tyFB.tyBtnRemoteClamp.bValue		:= FALSE;
		tyP0932MagConv3.tyFB.tyBtnRemoteUnclamp.bRtCompl	:= FALSE;
		tyP0932MagConv3.tyFB.tyBtnRemoteUnclamp.bValue		:= FALSE;

	END_IF

	//Mask
	IF p_eMagConv2Clp3Status = Error THEN

		fUIInRtStatOff(ADR(tyP0932MagConv3.tyDC.tyBtnMagIn.uiMaskRtStat));
		fUIInRtStatOff(ADR(tyP0932MagConv3.tyDC.tyBtnMagOut.uiMaskRtStat));
		fUIInRtStatOff(ADR(tyP0932MagConv3.tyDC.tyBtnFixedClamp.uiMaskRtStat));
		fUIInRtStatOff(ADR(tyP0932MagConv3.tyDC.tyBtnFixedUnclamp.uiMaskRtStat));
		fUIInRtStatOff(ADR(tyP0932MagConv3.tyDC.tyBtnRemoteClamp.uiMaskRtStat));
		fUIInRtStatOff(ADR(tyP0932MagConv3.tyDC.tyBtnRemoteUnclamp.uiMaskRtStat));

	ELSIF tyP0932MagConv3.tyDC.tyBtnMagIn.bValue = TRUE THEN

		fUIInRtStatHide(ADR(tyP0932MagConv3.tyDC.tyBtnMagIn.uiMaskRtStat));
		fUIInRtStatOff(ADR(tyP0932MagConv3.tyDC.tyBtnMagOut.uiMaskRtStat));
		fUIInRtStatOff(ADR(tyP0932MagConv3.tyDC.tyBtnFixedClamp.uiMaskRtStat));
		fUIInRtStatOff(ADR(tyP0932MagConv3.tyDC.tyBtnFixedUnclamp.uiMaskRtStat));
		fUIInRtStatOff(ADR(tyP0932MagConv3.tyDC.tyBtnRemoteClamp.uiMaskRtStat));
		fUIInRtStatOff(ADR(tyP0932MagConv3.tyDC.tyBtnRemoteUnclamp.uiMaskRtStat));

	ELSIF tyP0932MagConv3.tyDC.tyBtnMagOut.bValue = TRUE THEN

		fUIInRtStatOff(ADR(tyP0932MagConv3.tyDC.tyBtnMagIn.uiMaskRtStat));
		fUIInRtStatHide(ADR(tyP0932MagConv3.tyDC.tyBtnMagOut.uiMaskRtStat));
		fUIInRtStatOff(ADR(tyP0932MagConv3.tyDC.tyBtnFixedClamp.uiMaskRtStat));
		fUIInRtStatOff(ADR(tyP0932MagConv3.tyDC.tyBtnFixedUnclamp.uiMaskRtStat));
		fUIInRtStatOff(ADR(tyP0932MagConv3.tyDC.tyBtnRemoteClamp.uiMaskRtStat));
		fUIInRtStatOff(ADR(tyP0932MagConv3.tyDC.tyBtnRemoteUnclamp.uiMaskRtStat));

	ELSE

		fUIInRtStatHide(ADR(tyP0932MagConv3.tyDC.tyBtnMagIn.uiMaskRtStat));
		fUIInRtStatHide(ADR(tyP0932MagConv3.tyDC.tyBtnMagOut.uiMaskRtStat));
		fUIInRtStatHide(ADR(tyP0932MagConv3.tyDC.tyBtnFixedClamp.uiMaskRtStat));
		fUIInRtStatHide(ADR(tyP0932MagConv3.tyDC.tyBtnFixedUnclamp.uiMaskRtStat));
		fUIInRtStatHide(ADR(tyP0932MagConv3.tyDC.tyBtnRemoteClamp.uiMaskRtStat));
		fUIInRtStatHide(ADR(tyP0932MagConv3.tyDC.tyBtnRemoteUnclamp.uiMaskRtStat));

	END_IF

END_ACTION
```
